//testReal:=BYTE_TO_REAL(arr_RcvData_Temp);
//数据接收处理
reciveFtrig(CLK:=receive1.busy);
IF reciveFtrig.Q THEN
	arr_RcvDataString:=arr_RcvDataStringTemp;
	arr_RcvDataStringTemp:=arr_RcvDataStringClear;
	RcvDataFlag:=TRUE;
	serialConnected:=TRUE;
END_IF
recTon(IN:=RcvDataFlag, PT:=T#20MS);
IF recTon.Q THEN
	RcvDataFlag:=FALSE;
END_IF
againSendS3(IN:=NOT RcvDataFlag,PT:=T#5S);
IF againSendS3.Q THEN
	sendstr:='S3$R';
	serialExcute:=TRUE;
	serialConnected:=FALSE;
	againSendS3(IN:=FALSE);
END_IF
IF TRUE THEN
	IF BYTE_TO_INT(arr_RcvDataString[4]-48)>0 THEN
		rec_ManulOrAuto:=TRUE;
		rec_MAStr:='Manul';
	ELSE
		rec_ManulOrAuto:=FALSE;
		rec_MAStr:='Auto';
	END_IF
	// 公式：(AD_CH6-LD_MIN)*(100/(LD_MAX-LD_MIN))
	AD_CH6:=CalMeth(arr_RcvDataString[28])*16*16+CalMeth(arr_RcvDataString[29])*16+CalMeth(arr_RcvDataString[30]);
	load:=(INT_TO_REAL(AD_CH6)-INT_TO_REAL(R00_LDMIN))*(100.0/(INT_TO_REAL(R01_LDMAX)-INT_TO_REAL(R00_LDMIN)));
	IF load>100.0 THEN
		load:=100.0;
		loadRunErr:=TRUE;
	END_IF
	IF load<0.0 THEN
		load:=0.0;
		loadRunErr:=TRUE;
	END_IF
	IF load<100.0 AND load>=0.0 THEN
		loadRunErr:=FALSE;
	END_IF
	// 公式：(AD_CH7-PH_MIN)*(100/(PH_MAX-PH_MIN))
	AD_CH7:=CalMeth(arr_RcvDataString[31])*16*16+CalMeth(arr_RcvDataString[32])*16+CalMeth(arr_RcvDataString[33]);	
	phase:=(INT_TO_REAL(AD_CH7)-INT_TO_REAL(R02_PHMIN))*(100.0/(INT_TO_REAL(R03_PHMAX)-INT_TO_REAL(R02_PHMIN)));
	IF phase>100.0 THEN
		phase:=100.0;
		phashRunErr:=TRUE;
	END_IF
	IF phase<0.0 THEN
		phase:=0.0;
		phashRunErr:=TRUE;
	END_IF
	IF phase<100.0 AND phase>=0.0 THEN
		phashRunErr:=FALSE;
	END_IF
END_IF
ACT_Send();
ACT_SetPreset();

ACTION ACT_Send:

CASE serialStep OF
	0:
	IF serialExcute THEN
		serialExcute:=FALSE;
		IF NOT serialBusy THEN
			serialStep:=90;
			serialBusy:=TRUE;
			serialDone:=FALSE;
			serialError:=FALSE;
			serialTimeOut:=FALSE;
			serialRecError:=FALSE;
		END_IF
	END_IF
	Timer1(IN:= FALSE);
	;
	10:
		arr_SendData:='SPL$R';
		send1(
			pSendData:= ADR(arr_SendData), 
			Length:=INT_TO_UDINT(LEN(arr_SendData)), 
			Busy=> , 
			Error=> , 
			TXbuffer:= gTxBuffer_SRF);
		serialStep:=serialStep+1;
	11:
		Timer1(IN:= NOT timer1.q, PT:=T#10MS);
		IF Timer1.Q THEN
			serialStep:=serialStep+1;
			Timer1(IN:= FALSE);
		END_IF
	12:
		Timer1(IN:= NOT timer1.q, PT:=T#500MS);
		IF Timer1.Q THEN
			serialStep:=6000;
			Timer1(IN:= FALSE);
			serialTimeOut:=TRUE;
			RETURN;
		END_IF
		IF NOT send1.busy AND NOT RcvDataFlag THEN
			Timer1(IN:= FALSE);
			serialTimeOut:=FALSE;
			serialStep:=serialStep+1;
		END_IF
		IF send1.Error <> COMERROR_NOERROR THEN
			serialRecError:=TRUE;
		END_IF
	13:
		Timer1(IN:= NOT timer1.q, PT:=T#50MS);
		IF Timer1.Q THEN
			serialStep:=90;
			Timer1(IN:= FALSE);
		END_IF
	90:
		arr_SendData:=sendstr;
		serialStep:=100;
	100:
		send1(
			pSendData:= ADR(arr_SendData), 
			Length:= INT_TO_UDINT(LEN(arr_SendData)), 
			Busy=> , 
			Error=> , 
			TXbuffer:= gTxBuffer_SRF);
		serialStep:=serialStep+10;
	110:
		Timer1(IN:= NOT timer1.q, PT:=T#10MS);
		IF Timer1.Q THEN
			serialStep:=serialStep+10;
			Timer1(IN:= FALSE);
		END_IF
	120:
		Timer1(IN:= NOT timer1.q, PT:=T#500MS);
		IF Timer1.Q THEN
			serialStep:=6000;
			Timer1(IN:= FALSE);
			serialTimeOut:=TRUE;
			RETURN;
		END_IF
		IF NOT send1.busy  THEN
			Timer1(IN:= FALSE);
			serialTimeOut:=FALSE;
			serialStep:=200;
		END_IF
		IF send1.Error <> COMERROR_NOERROR THEN
			serialRecError:=TRUE;
		END_IF
	200://数据处理
		serialStep:=serialStep+10;
	210:
		Timer1(IN:= NOT timer1.q, PT:=T#10MS);
		IF Timer1.Q THEN
			serialStep:=serialStep+10;
			Timer1(IN:= FALSE);
		END_IF
	220:
		//数据转换
		Timer1(IN:= FALSE);
		serialStep:=1000;
	
	1000:
		Timer1(IN:= NOT timer1.q, PT:=T#50MS);
		IF Timer1.Q THEN
			serialStep:=5000;
			Timer1(IN:= FALSE);
			// sendstr:='';
			serialTimeOut:=FALSE;
		END_IF
	;
	5000://done
		serialBusy:=FALSE;
		serialDone:=TRUE;
		serialError:=FALSE;
		serialStep:=0;
	;
	6000://error
		serialBusy:=FALSE;
		serialDone:=FALSE;
		serialError:=TRUE;
		serialStep:=0;
	;
	
END_CASE
END_ACTION

ACTION ACT_SetPreset:
CASE setPresetStep OF
	0:
	IF setPresetExt THEN
		setPresetExt:=FALSE;
		IF NOT setPresetBusy THEN
			setPresetStep:=100;
			setPresetBusy:=TRUE;
			setPresetDone:=FALSE;
			setPresetError:=FALSE;
		END_IF
	END_IF
	TimerSetPreset(IN:= FALSE);
	;
	100:
		decimalvalue:=LREAL_TO_INT(goPosLoad*10);
		decimalvalueP:=LREAL_TO_INT(goPosPhase*10);
		hexString:='';
		hexStringP:='';
		sendstr:='';
		IF goPosLoad>100 OR goPosLoad<0 OR goPosPhase>100 OR goPosPhase<0 THEN
			;
		ELSE
			IF goPosLoad=0 THEN
				hexString:='000';
			ELSE
				index:=(decimalvalue/256);
				hexString:=CONCAT(hexString,hexChars[index]);
				index:=((decimalvalue-index*256)/16);
				hexString:=CONCAT(hexString,hexChars[index]);
				index:=(decimalvalue MOD 16);
				hexString:=CONCAT(hexString,hexChars[index]);
			END_IF
			IF goPosPhase=0 THEN
				hexStringP:='000';
			ELSE
				index:=(decimalvalueP/256);
				hexStringP:=CONCAT(hexStringP,hexChars[index]);
				index:=((decimalvalueP-index*256)/16);
				hexStringP:=CONCAT(hexStringP,hexChars[index]);
				index:=(decimalvalueP MOD 16);
				hexStringP:=CONCAT(hexStringP,hexChars[index]);
			END_IF
			sendstr:=CONCAT(sendstr,'$$APGR');
			sendstr:=CONCAT(sendstr,hexString);
			sendstr:=CONCAT(sendstr,hexStringP);
			sendstr:=CONCAT(sendstr,'$R');
			serialExcute:=TRUE;
		END_IF
		setPresetStep:=setPresetStep+10;
	110:
		TimerSetPreset(IN:= TRUE,PT:=T#0.1S);
		IF TimerSetPreset.Q THEN
			TimerSetPreset(IN:= FALSE);
			setPresetStep:=setPresetStep+10;
		END_IF
	120:
		IF serialDone AND NOT serialBusy AND 
		ABS(load-goPosLoad)<0.5 AND ABS(phase-goPosPhase)<0.5 THEN
			setPresetStep:=setPresetStep+10;
		END_IF
		IF serialError THEN
			setPresetStep:=6000;
			RETURN;
		END_IF
	130:
		sendstr:='';
		sendstr:='P0$R';
		serialExcute:=TRUE;
		setPresetStep:=setPresetStep+10;
	140:
		TimerSetPreset(IN:= TRUE,PT:=T#0.03S);
		IF TimerSetPreset.Q THEN
			TimerSetPreset(IN:= FALSE);
			setPresetStep:=setPresetStep+10;
		END_IF
	150:
		IF serialDone THEN
			setPresetStep:=5000;
		END_IF
	
	5000://done
		setPresetBusy:=FALSE;
		setPresetDone:=TRUE;
		setPresetError:=FALSE;
		DataSave.fbDataSaveModule_EX_1.setLrealValue(FuncModule_RS232_SRF.goPosLoad,1);
		DataSave.fbDataSaveModule_EX_1.setLrealValue(FuncModule_RS232_SRF.goPosPhase,2);
		DataSave.fbDataSaveModule_EX_1.saveB:=TRUE;
		ups_CX51X0.Act_Wrtie();
		setPresetStep:=0;
	;
	6000://error
		setPresetBusy:=FALSE;
		setPresetDone:=FALSE;
		setPresetError:=TRUE;
		setPresetStep:=0;
	;
	
END_CASE
END_ACTION

METHOD CalASII_Str : STRING
VAR_INPUT
	date1:UINT;
END_VAR
IF date1=10 THEN
	CalASII_Str:='A';
END_IF
IF date1=11 THEN
	CalASII_Str:='B';
END_IF
IF date1=12 THEN
	CalASII_Str:='C';
END_IF
IF date1=13 THEN
	CalASII_Str:='D';
END_IF
IF date1=14 THEN
	CalASII_Str:='E';
END_IF
IF date1=15 THEN
	CalASII_Str:='F';
END_IF
IF date1<10 THEN
	CalASII_Str:=UINT_TO_STRING(date1);
END_IF
IF date1>15 THEN
	CalASII_Str:=UINT_TO_STRING(date1);
END_IF
END_METHOD

METHOD CalMeth : INT
VAR_INPUT
	byteIn:BYTE;
END_VAR
VAR_OUTPUT
	outInt:INT;
END_VAR
IF byteIn>=48 AND byteIn<=57 THEN
	outInt:=byteIn-48;
ELSE
	outInt:=byteIn-65+10;
END_IF
CalMeth:=outInt;
END_METHOD

METHOD LoadAndPhaseGo : BOOL
VAR_INPUT
	
END_VAR
VAR_OUTPUT
	
END_VAR
setPresetExt:=TRUE;
END_METHOD

METHOD LoadDEC : BOOL
VAR_INPUT
END_VAR
sendstr:='J84$R';
serialExcute:=true;
END_METHOD

METHOD LoadINC : BOOL
VAR_INPUT
END_VAR
sendstr:='J85$R';
serialExcute:=true;
END_METHOD

METHOD ManulORAuto : BOOL
VAR_INPUT
END_VAR
IF NOT rec_ManulOrAuto THEN
	sendstr:='M$R';
	serialExcute:=TRUE;
ELSE
	sendstr:='L$R';
	serialExcute:=TRUE;
END_IF
END_METHOD

METHOD PhaseDEC : BOOL
VAR_INPUT
END_VAR
sendstr:='J48$R';
serialExcute:=true;
END_METHOD

METHOD PhaseINC : BOOL
VAR_INPUT
END_VAR
sendstr:='J58$R';
serialExcute:=true;
END_METHOD

END_PROGRAM

// ---- POUs/Data/DownTimeRecordPOU.TcPOU
PROGRAM DownTimeRecordPOU
VAR
	fbGetCurTaskIndex:GetCurTaskIndex;
	nTaskNo:INT;
	tonPush:TON;
	tPush:TIME:=T#59.9S;
	fDownTime:REAL;
	fOtherDownTime:REAL;
	fOpDownTime:REAL;
END_VAR
VAR
	stPowerOnTime:ST_DownTimeRecord;// 记录上电运行总时间，从开始自动到结束自动的时间
	nPowerOnDay:UDINT:=0;// 记录上电天数

	stAutoRunTime:ST_DownTimeRecord;// 记录自动运行总时间，从开始自动到结束自动的时间
	AutoRunTime_temp:LREAL;// 缓存时间
	
	stManualMachineDownTime:ST_DownTimeRecord;// 记录手动状态下设备DownTime，
	ManualMachineDownTime_temp:LREAL;// 缓存时间
	
	stMachineDownTime:ST_DownTimeRecord;// 记录设备DownTime，从报错上升沿到下降沿
	MachineDownTime_temp:LREAL;// 缓存时间
	
	stOtherDownTime:ST_DownTimeRecord;// 记录设备其他DownTime，从暂停上升沿到下降沿
	OtherDownTime_temp:LREAL;// 缓存时间
	
	stOpLoadDownTime:ST_DownTimeRecord;// 记录设备操作员上料DownTime，从动作超时上升沿到下降沿
	OpLoadDownTime_Fix:LREAL;// 操作员固定时间
	OpLoadDownTime_temp:LREAL;// 缓存时间
	
	stOpUnloadDownTime:ST_DownTimeRecord;// 记录设备操作员下料DownTime，从动作超时上升沿到下降沿
	OpUnloadDownTime_Fix:LREAL;// 操作员固定时间
	OpUnloadDownTime_temp:LREAL;// 缓存时间
	
END_VAR


// 记录PLC上电总时间
	fbGetCurTaskIndex(index=>nTaskNo);
	IF TwinCAT_SystemInfoVarList._TaskInfo[nTaskNo].FirstCycle THEN// 上电初始时间
		stPowerOnTime.startTime:=TIME();
		nPowerOnDay:=0;
		stManualMachineDownTime.startTime:=TIME();
		ManualMachineDownTime_temp:=0;
		
		initState(stAutoRunTime);
		initState(stManualMachineDownTime);
		initState(stMachineDownTime);
		initState(stOtherDownTime);
		initState(stOpLoadDownTime);
		initState(stOpUnloadDownTime);
	END_IF
	stPowerOnTime.endTime:=TIME();
	calcTime(stPowerOnTime);
	
	stPowerOnTime.bMonitor:=((stPowerOnTime.start2end_s>=3600));// 监控的状态
	stPowerOnTime.rTrig(CLK:=stPowerOnTime.bMonitor);
	IF stPowerOnTime.rTrig.Q THEN// 累加1天
		stPowerOnTime.startTime:=TIME();
		nPowerOnDay:=nPowerOnDay+1;
	END_IF

// 记录自动运行总时间
	stAutoRunTime.rTrig(CLK:=gAutoRunningFlag);
	IF stAutoRunTime.rTrig.Q THEN// 注意，在初进入自动时同步 startTime 和 endTime
		// 此次是否需要初始化？
		(*initState(stAutoRunTime);
		initState(stMachineDownTime);
		initState(stOtherDownTime);
		initState(stOpLoadDownTime);
		initState(stOpUnloadDownTime);*)
		
		stAutoRunTime.startTime:=TIME();
		//
	END_IF
	stAutoRunTime.fTrig(CLK:=gAutoRunningFlag);
	IF stAutoRunTime.fTrig.Q THEN// 注意，在初进入自动时同步 startTime 和 endTime
		stManualMachineDownTime.startTime:=TIME();
		ManualMachineDownTime_temp:=0;
		
		stAutoRunTime.endTime:=TIME();
		calcTime(stAutoRunTime);
		AutoRunTime_temp:=0;
		stAutoRunTime.record_s:=stAutoRunTime.start2end_s;
		
		(*calcTime(stMachineDownTime);
		calcTime(stOtherDownTime);
		calcTime(stOpLoadDownTime);
		calcTime(stOpUnloadDownTime);
		stMachineDownTime.record_s:=stMachineDownTime.start2end_s;
		stOtherDownTime.record_s:=stOtherDownTime.start2end_s;
		stOpLoadDownTime.record_s:=stOpLoadDownTime.start2end_s;
		stOpUnloadDownTime.record_s:=stOpUnloadDownTime.start2end_s;*)
		// 做时间记录
		
		// 此次是否需要初始化？
		(*initState(stAutoRunTime);
		initState(stMachineDownTime);
		initState(stOtherDownTime);
		initState(stOpLoadDownTime);
		initState(stOpUnloadDownTime);*)
	END_IF


// 记录自动运行下: MachineDownTime 时间; OtherDownTime 时间; OpLoadDownTime 时间;  OpUnLoadDownTime 时间; 
	IF gAutoRunningFlag THEN// 自动状态下
	 (*MachineDownTime*) // 报错 上升沿-下降沿
		stMachineDownTime.bMonitor:=(gRunningState=RunningStatus.eErrorState);// 监控的状态
		stMachineDownTime.rTrig(CLK:=stMachineDownTime.bMonitor);
		IF stMachineDownTime.rTrig.Q THEN// 记录开始时间
			stMachineDownTime.startTime:=TIME();
			MachineDownTime_temp:=0;
		END_IF
		IF stMachineDownTime.bMonitor THEN
			stMachineDownTime.endTime:=TIME();
			calcTime(stMachineDownTime);
			MachineDownTime_temp:=(stMachineDownTime.start2end_s)-MachineDownTime_temp;// 获取每个扫描周期产生的时间差
			stMachineDownTime.record_s:=stMachineDownTime.record_s+MachineDownTime_temp;
			MachineDownTime_temp:=(stMachineDownTime.start2end_s);// 缓存最后一个扫描周期的总时长
		END_IF
		stMachineDownTime.fTrig(CLK:=stMachineDownTime.bMonitor);
		IF stMachineDownTime.fTrig.Q THEN// 记录结束状态
			stMachineDownTime.endTime:=TIME();
			calcTime(stMachineDownTime);
			MachineDownTime_temp:=0;
			// 做时间记录
				(*
				gDownTimeLog.append(CONCAT('DT,stMachineDownTime,',TO_STRING(stMachineDownTime.record_s)));
				*)
		END_IF
	 //
	 (*OtherDownTime*) // 暂停 上升沿-下降沿
		stOtherDownTime.bMonitor:=(gRunningState=RunningStatus.ePauseState);// 监控的状态
		stOtherDownTime.rTrig(CLK:=stOtherDownTime.bMonitor);
		IF stOtherDownTime.rTrig.Q THEN// 记录开始时间
			stOtherDownTime.startTime:=TIME();
			OtherDownTime_temp:=0;
		END_IF
		IF stOtherDownTime.bMonitor THEN
			stOtherDownTime.endTime:=TIME();
			calcTime(stOtherDownTime);
			OtherDownTime_temp:=(stOtherDownTime.start2end_s)-OtherDownTime_temp;// 获取每个扫描周期产生的时间差
			stOtherDownTime.record_s:=stOtherDownTime.record_s+OtherDownTime_temp;
			OtherDownTime_temp:=(stOtherDownTime.start2end_s);// 缓存最后一个扫描周期的总时长
		END_IF
		stOtherDownTime.fTrig(CLK:=stOtherDownTime.bMonitor);
		IF stOtherDownTime.fTrig.Q THEN// 记录结束状态
			stOtherDownTime.endTime:=TIME();
			calcTime(stOtherDownTime);
			OtherDownTime_temp:=0;
			// 做时间记录
				(*
				gDownTimeLog.append(CONCAT('DT,stOtherDownTime,',TO_STRING(stOtherDownTime.record_s)));
				*)
		END_IF
	 //
	 (*OpLoadDownTime*) //  上升沿-下降沿
	 	// 此处不会记录第一次进入自动时，OP不上料的情况
//		stOpLoadDownTime.rTrig(CLK:=L_Robot_Load.Can_Getting_DUT);//(CLK:=L_Robot_Load.Getting_DUT);
//		IF stOpLoadDownTime.rTrig.Q OR (gRunningState<>RunningStatus.eAutoState) THEN// 记录开始时间
//			stOpLoadDownTime.startTime:=TIME();
//			OpLoadDownTime_temp:=0;
//			stOpLoadDownTime.bMonitor:=TRUE;
//		END_IF
//		IF stOpLoadDownTime.bMonitor THEN
//			stOpLoadDownTime.endTime:=TIME();
//			calcTime(stOpLoadDownTime);
//			OpLoadDownTime_Fix:=3;// 常数, 按实际情况配置------------------------------------------------------------------------------
//			IF (stOpLoadDownTime.start2end_s>OpLoadDownTime_Fix) THEN
//				OpLoadDownTime_temp:=(stOpLoadDownTime.start2end_s(*-OpLoadDownTime_Fix*))-OpLoadDownTime_temp;// 获取每个扫描周期产生的时间差
//				stOpLoadDownTime.record_s:=stOpLoadDownTime.record_s+OpLoadDownTime_temp;
//				OpLoadDownTime_temp:=(stOpLoadDownTime.start2end_s(*-OpLoadDownTime_Fix*));// 缓存最后一个扫描周期的总时长
//			END_IF
//		END_IF
//		stOpLoadDownTime.fTrig(CLK:=L_Robot_Load.Can_Getting_DUT);
//		IF stOpLoadDownTime.fTrig.Q THEN// 记录结束状态
//			stOpLoadDownTime.bMonitor:=FALSE;
//			stOpLoadDownTime.endTime:=TIME();
//			calcTime(stOpLoadDownTime);
//			OpLoadDownTime_temp:=0;// 清除缓存时间
//			// 做时间记录
//				(*
//				gDownTimeLog.append(CONCAT('DT,stOpLoadDownTime,',TO_STRING(stOpLoadDownTime.record_s)));
//				*)
//		END_IF
//	 //
//	 (*OpUnLoadDownTime*) //  上升沿-下降沿
//		stOpUnloadDownTime.bMonitor:=gStationUnLoad.I_BeltEndisHaveDutSensor_1 OR gStationUnLoad.I_BeltEndisHaveDutSensor_2;// 监控的状态
//		stOpUnloadDownTime.rTrig(CLK:=stOpUnloadDownTime.bMonitor);
//		IF stOpUnloadDownTime.rTrig.Q OR (gRunningState<>RunningStatus.eAutoState) THEN// 记录开始时间
//			stOpUnloadDownTime.startTime:=TIME();
//			OpUnloadDownTime_temp:=0;
//		END_IF
//		IF stOpUnloadDownTime.bMonitor THEN
//			stOpUnloadDownTime.endTime:=TIME();
//			calcTime(stOpUnloadDownTime);
//			OpUnloadDownTime_Fix:=3;// 常数, 按实际情况配置------------------------------------------------------------------------------
//			IF (stOpUnloadDownTime.start2end_s>OpUnloadDownTime_Fix) THEN
//				OpUnloadDownTime_temp:=(stOpUnloadDownTime.start2end_s(*-OpUnloadDownTime_Fix*))-OpUnloadDownTime_temp;// 获取每个扫描周期产生的时间差
//				stOpUnloadDownTime.record_s:=stOpUnloadDownTime.record_s+OpUnloadDownTime_temp;
//				OpUnloadDownTime_temp:=(stOpUnloadDownTime.start2end_s(*-OpUnloadDownTime_Fix*));// 缓存最后一个扫描周期的总时长
//			END_IF
//		END_IF
//		stOpUnloadDownTime.fTrig(CLK:=stOpUnloadDownTime.bMonitor);
//		IF stOpUnloadDownTime.fTrig.Q THEN// 记录结束状态
//			stOpUnloadDownTime.endTime:=TIME();
//			calcTime(stOpUnloadDownTime);
//			OpUnloadDownTime_temp:=0;// 清除缓存时间
//			// 做时间记录
//				(*
//				gDownTimeLog.append(CONCAT('DT,stOpUnloadDownTime,',TO_STRING(stOpUnloadDownTime.record_s)));
//				*)
//		END_IF
//	 //
	ELSE// 手动状态下
		stManualMachineDownTime.endTime:=TIME();
		calcTime(stManualMachineDownTime);
		ManualMachineDownTime_temp:=(stManualMachineDownTime.start2end_s)-ManualMachineDownTime_temp;// 获取每个扫描周期产生的时间差
		stManualMachineDownTime.record_s:=stManualMachineDownTime.record_s+ManualMachineDownTime_temp;
		ManualMachineDownTime_temp:=(stManualMachineDownTime.start2end_s);// 缓存最后一个扫描周期的总时长
	END_IF

// 定时上报
tonPush(IN:=NOT tonPush.Q,PT:=tPush);
IF tonPush.Q THEN
	IF gAutoRunningFlag THEN
		stAutoRunTime.endTime:=TIME();
		calcTime(stAutoRunTime);
		AutoRunTime_temp:=0;
		stAutoRunTime.record_s:=stAutoRunTime.start2end_s;
//		gPowerONTotalTime:=gPowerONTotalTime+1;
	END_IF
	fDownTime:=TO_REAL(stManualMachineDownTime.record_s+stMachineDownTime.record_s);
	fOtherDownTime:=TO_REAL(stOtherDownTime.record_s);
	fOpDownTime:=TO_REAL(stOpLoadDownTime.record_s+stOpUnloadDownTime.record_s);
	
	//(*
	gDownTimeLog.append(CONCAT('DT,stAutoRunTime,',TO_STRING(stAutoRunTime.record_s)));
	gDownTimeLog.append(CONCAT('DT,stManualMachineDownTime,',TO_STRING(stManualMachineDownTime.record_s)));
	gDownTimeLog.append(CONCAT('DT,stMachineDownTime,',TO_STRING(stMachineDownTime.record_s)));
	gDownTimeLog.append(CONCAT('DT,stOtherDownTime,',TO_STRING(stOtherDownTime.record_s)));
//	gDownTimeLog.append(CONCAT('DT,stOpLoadDownTime,',TO_STRING(stOpLoadDownTime.record_s)));
//	gDownTimeLog.append(CONCAT('DT,stOpUnloadDownTime,',TO_STRING(stOpUnloadDownTime.record_s)));
	//*)
	// 此次需要做发送给上位机的逻辑
//	PLC_SW1.appendSend(0,0,80,0.0,TO_REAL(stManualMachineDownTime.record_s),0.0,TO_REAL(stOtherDownTime.record_s),0.0,gErrIDToSW,'');
	
	// 记录完毕清除数据，重新记录
	initState(stAutoRunTime);
	initState(stManualMachineDownTime);
	initState(stMachineDownTime);
	initState(stOtherDownTime);
	initState(stOpLoadDownTime);
	initState(stOpUnloadDownTime);
	AutoRunTime_temp:=0;
	ManualMachineDownTime_temp:=0;
	MachineDownTime_temp:=0;
	OpLoadDownTime_temp:=0;
	OpUnloadDownTime_temp:=0;
END_IF

METHOD calcTime : BOOL
VAR_IN_OUT
	stDownTimeRecord:ST_DownTimeRecord;
END_VAR

stDownTimeRecord.start2end_time:=(stDownTimeRecord.endTime-stDownTimeRecord.startTime);
stDownTimeRecord.start2end_ms:=TO_UDINT(stDownTimeRecord.endTime-stDownTimeRecord.startTime);
stDownTimeRecord.start2end_s:=TO_LREAL(stDownTimeRecord.start2end_ms)*0.001;
//stDownTimeRecord.startTime:=stDownTimeRecord.endTime;

calcTime:=TRUE;
END_METHOD

METHOD initState : BOOL
VAR_IN_OUT
	stDownTimeRecord:ST_DownTimeRecord;
END_VAR

stDownTimeRecord.bMonitor:=FALSE;
stDownTimeRecord.startTime:=stDownTimeRecord.endTime:=TIME();
stDownTimeRecord.start2end_ms:=0;
stDownTimeRecord.start2end_s:=0;
stDownTimeRecord.start2end_time:=TO_TIME(0);
stDownTimeRecord.record_s:=0;
stDownTimeRecord.rTrig(CLK:=FALSE);
stDownTimeRecord.fTrig(CLK:=FALSE);

initState:=TRUE;
END_METHOD

END_PROGRAM

// ---- POUs/Data/FB_WStringSave.TcPOU
PROGRAM FB_WStringSave
VAR CONSTANT
	Maxlenght:INT:=100;
END_VAR

VAR_INPUT
	filter:WSTRING:=",";
	readTrig:BOOL;
	writeTrig:BOOL;
	savePath : T_MaxString;
END_VAR
VAR_OUTPUT
	nErrorId : UDINT;
	bError : BOOL;
	readDone:BOOL;
	saveDone:BOOL;
	readError:BOOL;
	saveError:BOOL;
END_VAR
VAR
	fbFileOpen:FB_FILEOPEN;
	fbFileClose:FB_FILECLOSE;
	fbFileGet:FB_FILEGETS;
	fbFilePut:FB_FILEPUTS;
	fbWriter:FB_FILEWRITE;

	hFile : UINT;
	sReadLine : T_MaxString;
	wsWriteLine : WSTRING(255); 
	sWriteLine : T_MaxString;
	wsReadLine : WSTRING(255);
	wsReadTemp : WSTRING(255);
	itemp:INT;
	inputArry: ARRAY [1..Maxlenght] OF WSTRING;
	outputArry: ARRAY [1..Maxlenght] OF WSTRING;
	findposstart	:INT;
	findposend		:INT;
	find_pos		:INT;
	recStrTemp		:WSTRING(255);
	nReadStep : UINT;
	nWriteStep : UINT;
END_VAR

readDone:=FALSE;
fbFileOpen(
	sNetId:= , 
	sPathName:= , 
	nMode:= , 
	ePath:= , 
	bExecute:= , 
	tTimeout:= , 
	bBusy=> , 
	bError=> , 
	nErrId=> , 
	hFile=>hFile );
	
fbFileClose(
	sNetId:= , 
	hFile:= hFile, 
	bExecute:= , 
	tTimeout:= , 
	bBusy=> , 
	bError=> , 
	nErrId=> );

fbFileGet(
	sNetId:= , 
	hFile:= hFile, 
	bExecute:= , 
	tTimeout:= , 
	bBusy=> , 
	bError=> , 
	nErrId=> , 
	sLine=> , 
	bEOF=> );
	
fbFilePut(
	sNetId:= , 
	hFile:= hFile, 
	sLine:= , 
	bExecute:= , 
	tTimeout:= , 
	bBusy=> , 
	bError=> , 
	nErrId=> );
IF readTrig THEN
	nReadStep:=10;
	readTrig:=FALSE;
END_IF
IF writeTrig THEN
	nWriteStep:=10;
	writeTrig:=FALSE;
END_IF
Act_Read();
Act_Write();

ACTION Act_Read:
CASE nReadStep OF
	0:
	;
	10:
		//复位状态
		bError := FALSE;
		nErrorId := 0;
		fbFileopen(bExecute:= FALSE);
		fbFileclose(bExecute:= FALSE);
		fbFileGet(bExecute:= FALSE);
		readError:=FALSE;
		nReadStep := 20;
		fbFileopen(sNetId:= , sPathName:= savePath,ePath:= PATH_GENERIC, bExecute:= TRUE, nMode:=FOPEN_MODEREAD ,hFile=>hFile );
	20:	
		IF NOT fbFileopen.bBusy THEN
			fbFileopen(bExecute:= FALSE);
			IF fbFileopen.bError THEN//出错
				bError := TRUE;
				nErrorId := fbFileopen.nErrId;
				nReadStep := 200;
				readError:=TRUE;
			ELSE //正常
				
				nReadStep := 30;
			
			END_IF
		END_IF
	30:
		nReadStep := 40;
	40:
		nReadStep := 100;
	100:
		fbFileGet(hFile:= hFile, bExecute:= TRUE, sLine=>sReadLine);
		UTF8_TO_WSTRING(ADR(wsReadLine),ADR(sReadLine),SIZEOF(sReadLine));
		IF NOT fbFileGet.bBusy THEN
			fbFileGet(bExecute:= FALSE);
			IF fbFileGet.bError THEN//出错
				bError := TRUE;
				nErrorId := fbFileGet.nErrId;
				nReadStep := 200;
				readError:=TRUE;
			ELSE //正常
				IF NOT fbFileGet.bEOF THEN //继续读取
					nReadStep := 110;
				ELSE
					//读取完成
					nReadStep := 110;
				END_IF
				
				
			
			END_IF
		END_IF
		
	110:
		wsReadTemp:=wsReadLine;
		ReadToOut();
		nReadStep := 200;		
		;
	200:
		fbFileClose( hFile:= hFile, bExecute:= TRUE ,nErrId=> );
		IF NOT fbFileClose.bBusy THEN
			fbFileClose(bExecute:= FALSE);
			IF fbFileClose.bError THEN//出错
				bError := TRUE;
				nErrorId := fbFileClose.nErrId;
				nReadStep := 1000;
			ELSE //正常
				
				nReadStep := 2000;
			
			END_IF
		END_IF
		
	1000:
		//报错
		nReadStep := 0;
		
	2000:
		//完成
		nReadStep := 0;
		readDone:=TRUE;
END_CASE
END_ACTION

ACTION Act_Write:
CASE nWriteStep OF
	0:
	;
	10:
		//复位状态
		bError := FALSE;
		nErrorId := 0;
		fbFileOpen(bExecute:= FALSE);
		fbFileClose(bExecute:= FALSE);
		fbFilePut(bExecute:= FALSE);
		saveError:=FALSE;
		nWriteStep := 20;
	20:
		fbFileOpen(sNetId:= , sPathName:= savePath, nMode:= FOPEN_MODEWRITE, ePath:= , bExecute:= TRUE,hFile=>hFile );		
		IF NOT fbFileOpen.bBusy THEN
			fbFileOpen(bExecute:= FALSE);
			IF fbFileOpen.bError THEN//出错
				bError := TRUE;
				nErrorId := fbFileOpen.nErrId;
				nWriteStep := 200;
				saveError:=TRUE;
			ELSE //正常
				
				nWriteStep := 100;
			
			END_IF
		END_IF

	100:
		InToWrite();
		nWriteStep := 110;
	110:
		WSTRING_TO_UTF8(ADR(sWriteLine),ADR(wsWriteLine),SIZEOF(wsWriteLine));
		fbFilePut(hFile:= hFile, bExecute:= TRUE, sLine:=sWriteLine);
		
		IF NOT fbFilePut.bBusy THEN
			fbFilePut(bExecute:= FALSE);
			IF fbFilePut.bError THEN//出错
				bError := TRUE;
				nErrorId := fbFilePut.nErrId;
				nWriteStep := 200;
				saveError:=TRUE;
			ELSE //正常
				//写入完成
				nWriteStep := 200;	
			END_IF
		END_IF
		wsWriteLine:="";
				
		;
	200:
		fbFileClose( hFile:= hFile, bExecute:= TRUE ,nErrId=> );
		IF NOT fbFileClose.bBusy THEN
			fbFileClose(bExecute:= FALSE);
			IF fbFileClose.bError THEN//出错
				bError := TRUE;
				nErrorId := fbFileClose.nErrId;
				nWriteStep := 1000;
				saveError:=TRUE;
			ELSE //正常
				
				nWriteStep := 2000;
			
			END_IF
		END_IF
		
	1000:
		//报错
		nWriteStep := 0;
		
	2000:
		//完成
		nWriteStep := 0;
		
END_CASE
END_ACTION

METHOD getWString : BOOL
VAR_IN_OUT
	value:WSTRING;
END_VAR
VAR_INPUT
	num:UDINT;
END_VAR
IF 0<=num AND UDINT_TO_INT(num)<=Maxlenght THEN
	value:=outputArry[num];
	getWString:=TRUE;
ELSE
	value:="";
	getWString:=FALSE;
END_IF
END_METHOD

ACTION InToWrite:
FOR itemp:=1 TO Maxlenght DO
	wsWriteLine:=WCONCAT(wsWriteLine,inputArry[itemp]);
	wsWriteLine:=WCONCAT(wsWriteLine,filter);
END_FOR
END_ACTION

ACTION ReadToOut:
FOR itemp:=1 TO Maxlenght DO
	find_pos:=wFIND(wsReadTemp, filter);
	IF find_pos>0 THEN
		findposstart:=find_pos;
		outputArry[itemp]:=WMID(wsReadTemp,find_pos-1,1);
		wsReadTemp:=WDELETE(wsReadTemp,find_pos,1);
		find_pos:=0;
	END_IF
END_FOR
END_ACTION

METHOD setWString : BOOL
VAR_INPUT
	value:WSTRING;
END_VAR
VAR_INPUT
	num:UDINT;
END_VAR
IF 0<=num AND uDINT_TO_INT(num)<=Maxlenght THEN
	inputArry[num]:=value;
	setWString:=TRUE;
ELSE
	setWString:=FALSE;
END_IF
END_METHOD

END_PROGRAM

// ---- POUs/IO/TesterIO.TcPOU
{attribute'TcContextName':='IOTask'}
PROGRAM TesterIO
VAR
	fbIOBase_Input:FB_IOBase_Input_New;//工站1 Input 
	
	fbIOBase_Output:FB_IOBase_Output_New;//工站1 Output 
	 
	DOE_DOE1IO AT%I*:UDINT;
	DOE_DOE2IO AT%I*:UDINT;

	I_Handle1FixVacuum2Ext: INT;
	I_Handle1FixVacuum1Ext: INT;
END_VAR


//工站1 Input 
	fbIOBase_Input(
		iIOModuleNum:= 5, 
		iLanguage:= TO_UINT(gCNErrShow), //TO_UINT(gCNErrShow)
		sFileName:= 'C:\IOFilePath\Input1.csv', 
		bReload:= , 
		stIOBase=> );


//工站1 Output 
	fbIOBase_Output(
		iIOModuleNum:= 5, 
		stIOBase:= , 
		iLanguage:= TO_UINT(gCNErrShow), //TO_UINT(gCNErrShow)
		sFileName:= 'C:\IOFilePath\Output1.csv', 
		bReload:= );




//输入映射---映射到程序内部变量
ACT_Input();//工站1 Input 


//输出映射---映射到程序内部变量
ACT_Output();//工站1 Output 


// 通讯IO
ACT_Communication();

ACTION ACT_Communication:
FuncModule_RS232_TBP(
	noRotation=> gICP.TruboPumNoRotation, 
	brake=> gICP.TruboPumDcc, 
	acc=> gICP.TruboPumAcc, 
	atTagetSpeed=> gICP.TruboPumNormal, 
	alarm=> gICP.TruboPumAlarm, 
	remote=> gICP.TruboPumRemote, 
	failure=> gICP.TruboPumError, 
	rotationSpeed=> gICP.TruboPumRotationSpeed, 
	tMSTemperature=> gICP.TruboPumTMS);
END_ACTION

ACTION ACT_Input:
//(*驱动器DI 映射*)
//********************上料电机

//gLoad_AXIS.I_X1NLimit:=Load_X1IO.19;
//gLoad_AXIS.I_X1Home:=Load_X1IO.20;
//gLoad_AXIS.I_X1PLimit:=Load_X1IO.18;


//********************载具电机

//gTestSocket_AXIS.I_X1NLimit:=TestSocket_X1IO.18;
//gTestSocket_AXIS.I_X1Home:=TestSocket_X1IO.16;
//gTestSocket_AXIS.I_X1PLimit:=TestSocket_X1IO.17;

//gRXTest_AXIS.I_CY3NLimit:=RXTest_CY3IO.19;
//gRXTest_AXIS.I_CY3Home:=RXTest_CY3IO.22;
//gRXTest_AXIS.I_CY3PLimit:=RXTest_CY3IO.18;

//********************TX电机***********
////*******此处为量产660系列映射地址
//gTXTest_Axis.I_Y1NLimit:=TXTest_Y1IO.17;
//gTXTest_Axis.I_Y1Home:=TXTest_Y1IO.18;
//gTXTest_Axis.I_Y1PLimit:=TXTest_Y1IO.16;

/////////以下为临时应用 采用620驱动器///
//gTXTest_Axis.I_Y1NLimit:=TXTest_Y1IO.21;
//gTXTest_Axis.I_Y1Home:=TXTest_Y1IO.18;
//gTXTest_Axis.I_Y1PLimit:=TXTest_Y1IO.20;

//********************机台IO
//////模块1
//gDOE_AXIS.I_DOE2PLimit:=fbIOBase_Input.stIOBase[1].io[1]; //启动
//gDOE_AXIS.I_DOE2NLimit:=fbIOBase_Input.stIOBase[1].io[2]; //停止
//gMachineUtility.I_Reset:=fbIOBase_Input.stIOBase[1].io[3]; //复位
//gMachineUtility.I_EStop:=fbIOBase_Input.stIOBase[1].io[4] ; //急停
////:=fbIOBase_Input.stIOBase[1].io[5] ; //备用

////:=fbIOBase_Input.stIOBase[1].io[8] ; //备用
//gMachineUtility.I_PressureDetection1:=fbIOBase_Input.stIOBase[1].io[9] ; //气压检测

//gMachineUtility.I_SafeDoor_1:=fbIOBase_Input.stIOBase[1].io[13]; //安全门
//gMachineUtility.I_SafeDoor_2:=fbIOBase_Input.stIOBase[1].io[14]; //安全门
//gMachineUtility.I_SafeDoor_3:=fbIOBase_Input.stIOBase[1].io[15]; //安全门
//gMachineUtility.I_SafeDoor_4:=fbIOBase_Input.stIOBase[1].io[16]; //安全门


gICP.LiftPinExtSensor:=fbIOBase_Input.stIOBase[1].io[1]; //Lift UP
gICP.LiftPinRetSensor:=fbIOBase_Input.stIOBase[1].io[2]; //Lift Down
gICP.ElectrodeCylExtSensor:=fbIOBase_Input.stIOBase[1].io[3] AND fbIOBase_Input.stIOBase[1].io[4] AND fbIOBase_Input.stIOBase[1].io[14] AND fbIOBase_Input.stIOBase[1].io[15]; //Eletrode UP1 AND UP2
gICP.ElectrodeCylRetSensor:=fbIOBase_Input.stIOBase[1].io[5] AND fbIOBase_Input.stIOBase[1].io[6] AND fbIOBase_Input.stIOBase[1].io[16] AND fbIOBase_Input.stIOBase[2].io[1] ; //Eletrode Down1 AND Down2
gICP.GateDoorExtSensor:=fbIOBase_Input.stIOBase[1].io[7]; //GateDoor open
gICP.GateDoorRetSensor:=fbIOBase_Input.stIOBase[1].io[8]; //GateDoor Close
gICP.I_ARMHome:=fbIOBase_Input.stIOBase[1].io[9]; //ARM IN Sensor
gICP.I_LLSwitch:=fbIOBase_Input.stIOBase[1].io[10]; // LoadLock Switch Sensor
gICP.I_WaferCheck:=fbIOBase_Input.stIOBase[1].io[11]; //WaferCheck Sensor
gICP.PDVOpenSensor:=fbIOBase_Input.stIOBase[1].io[12]; //PDVOpen Sensor
gICP.PDVCloseSensor:=fbIOBase_Input.stIOBase[1].io[13]; //PDVClose Sensor
//gICP.PDV:=fbIOBase_Input.stIOBase[1].io[13]; //WaferCheck Sensor
//gICP.TruboPumAcc:=fbIOBase_Input.stIOBase[1].io[15]; // TruboPumAcc
//gICP.TruboPumDcc:=fbIOBase_Input.stIOBase[1].io[16]; // TruboPumDcc
//gICP.TruboPumNormal:=fbIOBase_Input.stIOBase[2].io[1]; // TruboPumNormal
gICP.I_ATMSensor:=fbIOBase_Input.stIOBase[2].io[2]; // ATMSensor
gICP.MachianicalPumAcc:=fbIOBase_Input.stIOBase[2].io[3]; // I_MP Start
gICP.MachianicalPumAlm:=fbIOBase_Input.stIOBase[2].io[4]; // I_MP Failure

gICP.PowerRF_Alrm:=fbIOBase_Input.stIOBase[2].io[5]; // 600W
gICP.SourceRF_Alrm:=fbIOBase_Input.stIOBase[2].io[6]; // 2000W
gICP.PowerRF_ON:=fbIOBase_Input.stIOBase[2].io[7]; // 600W
gICP.SourceRF_ON:=fbIOBase_Input.stIOBase[2].io[8]; // 2000W

 
gICP.I_WaterTemperatureCheck:=fbIOBase_Input.stIOBase[2].io[9]; 
gICP.I_WaterFlowCheck:=fbIOBase_Input.stIOBase[2].io[10];
gICP.I_PressureCheck:=fbIOBase_Input.stIOBase[2].io[11]; 
gICP.HeCheckGaugeReal:=PLC_HeliumPressure.bRecReal;
END_ACTION

ACTION ACT_Output:

//(*IO模块 映射*)
//模块1
fbIOBase_Output.stIOBase[1].io[1]:=gICP.ForlinLineValveExtRelay;
fbIOBase_Output.stIOBase[1].io[2]:=gICP.ISOExtRelay;
fbIOBase_Output.stIOBase[1].io[3]:=gICP.RoughValveExtRelay;
fbIOBase_Output.stIOBase[1].io[4]:=gICP.VentExtRelay;
fbIOBase_Output.stIOBase[1].io[5]:=gICP.SlowPummingExtRelay;
fbIOBase_Output.stIOBase[1].io[6]:=gICP.FastPummingExtRelay;
fbIOBase_Output.stIOBase[1].io[7]:=gICP.LiftPinRetRelay;
fbIOBase_Output.stIOBase[1].io[8]:=gICP.LiftPinExtRelay;
fbIOBase_Output.stIOBase[1].io[9]:=gICP.ElectrodeCylRetRelay;
fbIOBase_Output.stIOBase[1].io[10]:=gICP.ElectrodeCylExtRelay;
fbIOBase_Output.stIOBase[1].io[11]:=gICP.AIMExtRelay;
fbIOBase_Output.stIOBase[1].io[12]:=gICP.HeINExtRelay;
fbIOBase_Output.stIOBase[1].io[13]:=gICP.HePumExtRelay;
fbIOBase_Output.stIOBase[1].io[14]:=gICP.PDVOpenRelay;
fbIOBase_Output.stIOBase[1].io[15]:=gICP.PDVCloseRelay;
//fbIOBase_Output.stIOBase[1].io[16]:=gICP.PowerRFOpenRelay;
//模块2
fbIOBase_Output.stIOBase[2].io[1]:=gICP.MachianicalPumOpen;
//fbIOBase_Output.stIOBase[2].io[2]:=gICP.MachianicalPumOpen;// reset

fbIOBase_Output.stIOBase[2].io[3]:=gICP.GateDoorExtRelay;
fbIOBase_Output.stIOBase[2].io[4]:=gICP.GateDoorRetRelay;
//fbIOBase_Output.stIOBase[2].io[5]:=gICP.TruboPumOpen;
//fbIOBase_Output.stIOBase[2].io[6]:=gICP.TruboPumOpen;
//fbIOBase_Output.stIOBase[2].io[5]:=gICP.PowerRFResetRelay;
//fbIOBase_Output.stIOBase[2].io[6]:=gICP.SourceRFResetRelay;
//fbIOBase_Output.stIOBase[2].io[7]:=gICP.TruboPumReset;
fbIOBase_Output.stIOBase[2].io[8]:=gICP.SourceRFOpenRelay;
fbIOBase_Output.stIOBase[2].io[9]:=gICP.GVA1ExtRelay;
fbIOBase_Output.stIOBase[2].io[10]:=gICP.GVA2ExtRelay;
fbIOBase_Output.stIOBase[2].io[11]:=gICP.GVA3ExtRelay;
fbIOBase_Output.stIOBase[2].io[12]:=gICP.GVA4ExtRelay;
fbIOBase_Output.stIOBase[2].io[13]:=gICP.GVA5ExtRelay;
fbIOBase_Output.stIOBase[2].io[14]:=gICP.GVA6ExtRelay;
fbIOBase_Output.stIOBase[2].io[15]:=gICP.GVA7ExtRelay;
fbIOBase_Output.stIOBase[2].io[16]:=gICP.GVA8ExtRelay;

fbIOBase_Output.stIOBase[3].io[1]:=gICP.GVB1ExtRelay;
fbIOBase_Output.stIOBase[3].io[2]:=gICP.GVB2ExtRelay;
fbIOBase_Output.stIOBase[3].io[3]:=gICP.GVB3ExtRelay;
fbIOBase_Output.stIOBase[3].io[4]:=gICP.GVB4ExtRelay;
fbIOBase_Output.stIOBase[3].io[5]:=gICP.GVB5ExtRelay;
fbIOBase_Output.stIOBase[3].io[6]:=gICP.GVB6ExtRelay;
fbIOBase_Output.stIOBase[3].io[7]:=gICP.GVB7ExtRelay;
fbIOBase_Output.stIOBase[3].io[8]:=gICP.GVB8ExtRelay;
fbIOBase_Output.stIOBase[3].io[9]:=gICP.GVA9ExtRelay;
fbIOBase_Output.stIOBase[3].io[10]:=gICP.GVB9ExtRelay;
fbIOBase_Output.stIOBase[3].io[11]:=gICP.GVA10ExtRelay_Vent;
fbIOBase_Output.stIOBase[3].io[12]:=gICP.GV20ExtRelay_Main;
END_ACTION

END_PROGRAM

// ---- POUs/BaseModule/IO/FB_IOBase_Input_New.TcPOU
FUNCTION_BLOCK FB_IOBase_Input_New
VAR CONSTANT
	MAX_IO_MODULE_NUM:DINT:=15;
END_VAR
VAR_INPUT
	iIOModuleNum:DINT;//输入输出模块数量
	iLanguage:UINT;//0：英文；1：中文
	sFileName:T_MaxString:='C:\IOFilePath\iocsvfile.csv';//'Hard Disk\IOFilePath\iocsvfile.csv'
	bReload:BOOL;//加载配置文件 触发
END_VAR
VAR_OUTPUT
	stIOBase:ARRAY [1..MAX_IO_MODULE_NUM] OF ST_INPUT_IO;
END_VAR
VAR
	HMIITF:ST_IOBase_Show_HMI;
	
	iIOModuleNum_Temp:DINT;//输入输出模块数量
	
	next_R_TRIG:R_TRIG;
	back_R_TRIG:R_TRIG;
	targer_R_TRIG:R_TRIG;
	
	iCurrPage:DINT:=1;
	iIndex_1:DINT;
	iIndex_2:DINT;
	
	readBuff:ARRAY [1..MAX_IO_MODULE_NUM*16] OF ST_DataFmtBase;
	fbFileReadWrite:FB_IOFileReadWrite;
	bInit:BOOL;
	bRefresh:BOOL;
	Refresh_R_TRIG:R_TRIG;
	iLanguage_temp:UINT;//0：英文；1：中文
END_VAR


HMIITF.sIOType:='Input';

iIOModuleNum_Temp:=iIOModuleNum;
IF iIOModuleNum<0 THEN
	iIOModuleNum_Temp:=0;
ELSIF iIOModuleNum>MAX_IO_MODULE_NUM THEN
	iIOModuleNum_Temp:=MAX_IO_MODULE_NUM;
END_IF

(*HMI process*)
 (* Next button *)
	next_R_TRIG(CLK:=HMIITF.bNextPage);
	IF next_R_TRIG.Q THEN
		iCurrPage:=iCurrPage+1;
		bRefresh:=TRUE;
	END_IF
 (* Back button *)
	back_R_TRIG(CLK:=HMIITF.bBackPage);
	IF back_R_TRIG.Q THEN
		iCurrPage:=iCurrPage-1;
		bRefresh:=TRUE;
	END_IF
 (* Targer button *)
 	IF HMIITF.iTargerPage<=0 THEN
		HMIITF.iTargerPage:=iIOModuleNum_Temp;
	ELSIF HMIITF.iTargerPage>iIOModuleNum_Temp THEN
		HMIITF.iTargerPage:=1;
	END_IF
	targer_R_TRIG(CLK:=HMIITF.bTargerPage);
	IF targer_R_TRIG.Q THEN
		iCurrPage:=HMIITF.iTargerPage;
		bRefresh:=TRUE;
	END_IF

	IF iCurrPage<=0 THEN
		iCurrPage:=iIOModuleNum_Temp;
	ELSIF iCurrPage>iIOModuleNum_Temp THEN
		iCurrPage:=1;
	END_IF
	HMIITF.iCurrPage:=iCurrPage;
	HMIITF.iMaxPage:=iIOModuleNum_Temp;
	
	FOR iIndex_1:=1 TO 16 BY 1 DO
		HMIITF.bIO[iIndex_1]:=stIOBase[iCurrPage].io[iIndex_1];//IO状态映射
	END_FOR
	IF bRefresh THEN
		FOR iIndex_1:=1 TO 16 BY 1 DO
			HMIITF.bIO[iIndex_1]:=stIOBase[iCurrPage].io[iIndex_1];//IO状态映射
			
			CASE iLanguage OF
				0:
					FOR iIndex_2:=1 TO (MAX_IO_MODULE_NUM*16) BY 1 DO
						IF iCurrPage=readBuff[iIndex_2].nGroup AND iIndex_1=readBuff[iIndex_2].nNumber THEN
							HMIITF.sInfor[iIndex_1]:=TO_WSTRING(readBuff[iIndex_2].sTxt_ENG);
							IF 16=iIndex_1 THEN
								EXIT;
							END_IF
						END_IF
					END_FOR
				1:
					FOR iIndex_2:=1 TO (MAX_IO_MODULE_NUM*16) BY 1 DO
						IF iCurrPage=readBuff[iIndex_2].nGroup AND iIndex_1=readBuff[iIndex_2].nNumber THEN
							HMIITF.sInfor[iIndex_1]:=readBuff[iIndex_2].sTxt_CHN;
							IF 16=iIndex_1 THEN
								EXIT;
							END_IF
						END_IF
					END_FOR
			END_CASE
		END_FOR
	END_IF
	bRefresh:=FALSE;
	
(*Read csv file*)
	IF NOT bInit THEN
		bInit:=TRUE;
		bReload:=TRUE;
	END_IF
	fbFileReadWrite(
		readBuff:= readBuff, 
		sFileName:= sFileName, 
		bRead:= bReload, 
		sTxtHead:= 'GROUP,NUM,ENG,CHN,NO USE', 
		bBusy=> , 
		bDone=> , 
		bError=> , 
		nErrid=> );
	IF bReload THEN
		bReload:=FALSE;
	END_IF
	Refresh_R_TRIG(CLK:=fbFileReadWrite.bDone);
	IF Refresh_R_TRIG.Q THEN
		bRefresh:=TRUE;
	END_IF

END_FUNCTION_BLOCK

// ---- POUs/BaseModule/IO/ReadWriteCSV/FB_IOFileReadWrite.TcPOU
FUNCTION_BLOCK FB_IOFileReadWrite
VAR_IN_OUT
	readBuff:ARRAY [*] OF ST_DataFmtBase;
END_VAR
VAR_INPUT
	sFileName:T_MaxString:='C:\CsvFilePath\csvfile.csv';//'Hard Disk\CsvFilePath\csvfile.csv'
	bRead:BOOL;
	sTxtHead:STRING:='GROUP,NUM,ENG,CHN,NO USE';
END_VAR
VAR_OUTPUT
	bBusy:BOOL;
	bDone:BOOL;
	bError:BOOL;
	nErrid:UDINT;
END_VAR
VAR
	fbFileOpen:FB_FileOpen;
	fbFileClose:FB_FileClose;
	fbFileGets:FB_FileGets;
	fbReader:FB_CSVMemBufferReader;
	hFile:UINT:= 0;
	
	sReadLine:STRING(255);
	bReadEOF:BOOL;
	nReadCount:DINT;
	
	nStepRead:UINT;
	nReadBuffMin:DINT;
	nReadBuffMax:DINT;
	nReadBuffLen:DINT;
END_VAR


nReadBuffMin:=LOWER_BOUND(readBuff,1);//获取不定长数组的最小下标
nReadBuffMax:=UPPER_BOUND(readBuff,1);//获取不定长数组的最大下标
nReadBuffLen:=nReadBuffMax-nReadBuffMin+1;//获取数组有效长度

readCSV();

//

METHOD PRIVATE createDir : BOOL
VAR
	sPathNameTemp	: T_MaxString := 'C:\TwinCAT\Data.txt';
	sDriveTemp		: STRING(3);
	sDirTemp		: T_MaxString;
	sFileNameTemp	: T_MaxString;
	sExtTemp		: T_MaxString;
	bSuccess		: BOOL;
	fbCreateDir		: FB_CreateDir;
	sFileDirTemp	: T_MaxString;
END_VAR
sPathNameTemp:=sFileName;
bSuccess := F_SplitPathName(sPathName:= sPathNameTemp,
						sDrive:= sDriveTemp,
						sDir:= sDirTemp,
						sFileName:= sFileNameTemp,
						sExt:= sExtTemp );
IF bSuccess THEN
	bSuccess:=FALSE;
	IF LEFT(sDirTemp,LEN(sDirTemp)-1)<>'' THEN
		sFileDirTemp:=CONCAT(STR1:=sDriveTemp,STR2:=LEFT(sDirTemp,LEN(sDirTemp)-1));
		fbCreateDir(
			sNetId:= , 
			sPathName:= sFileDirTemp, 
			ePath:= PATH_GENERIC, 
			bExecute:= TRUE, 
			tTimeout:= , 
			bBusy=> , 
			bError=> , 
			nErrId=> );
	END_IF
END_IF
fbCreateDir(
	sNetId:= , 
	sPathName:= , 
	ePath:= , 
	bExecute:= FALSE, 
	tTimeout:= , 
	bBusy=> , 
	bError=> , 
	nErrId=> );
END_METHOD

METHOD PRIVATE readCSV : BOOL
VAR_INPUT
END_VAR
VAR
	nTemp_readCSV:INT;
	sGetValue_temp:STRING(255);
	bRtn:BOOL;
	nTemp1:INT;
END_VAR
DEFAULT_CSV_FIELD_SEP:= 16#2C;  //配置CSV文件的分割符，16#2C表明各个参数之间是用逗号分隔的。

CASE nStepRead OF
	0:
		IF bRead THEN
			bRead:=FALSE;
			bBusy:=TRUE;
			bDone:=FALSE;
			bError:=FALSE;
			nErrid:=0;
			
			nReadCount:=nReadBuffMin;			
			MEMSET(readBuff,0,TO_UDINT(SIZEOF(readBuff[nReadCount])*nReadBuffLen));//清空内存
			nStepRead:=100;
		END_IF
	100:
		fbFileOpen(bExecute:=FALSE);
		nStepRead:=nStepRead+10;
	110:
		fbFileOpen(
			sNetId:= , 
			sPathName:= sFileName, 
			nMode:= FOPEN_MODEREAD OR FOPEN_MODETEXT, 
			ePath:= PATH_GENERIC, 
			bExecute:= TRUE, 
			tTimeout:= , 
			bBusy=> , 
			bError=> , 
			nErrId=> , 
			hFile=> hFile);
		IF NOT fbFileOpen.bBusy THEN
			IF NOT fbFileOpen.bError THEN
				nStepRead:=nStepRead+10;
			ELSE
				nErrid:=fbFileOpen.nErrId;
				nStepRead:=60000;//Error
			END_IF
		END_IF
	120:
		fbFileGets(bExecute:=FALSE);
		IF nReadCount>nReadBuffMax THEN
			nStepRead:=150;
		ELSE
			nStepRead:=nStepRead+10;
		END_IF
	130:
		fbFileGets(
			sNetId:= , 
			hFile:= hFile, 
			bExecute:= TRUE, 
			tTimeout:= , 
			bBusy=> , 
			bError=> , 
			nErrId=> , 
			sLine=> sReadLine, 
			bEOF=> bReadEOF);
		IF NOT fbFileGets.bBusy THEN
			IF NOT fbFileGets.bError THEN
				sReadLine:=CONCAT(STR1:=sReadLine,STR2:='$R$L');
				nStepRead:=nStepRead+10;
			ELSE
				nErrid:=fbFileGets.nErrId;
				nStepRead:=60000;//Error
			END_IF
		END_IF
	140:
		IF ''<>sTxtHead AND FIND(sReadLine,sTxtHead)>0 THEN
			nStepRead:=120;
			RETURN;
		END_IF
		nTemp1:=0;
		fbReader.eCmd:=eEnumCmd_First;(* Read first field value *)
		FOR nTemp_readCSV:=0 TO 3 DO
			fbReader(
				eCmd:= , 
				pBuffer:= ADR(sReadLine), 
				cbBuffer:= SIZEOF(sReadLine), 
				bOk=> , 
				getValue=> sGetValue_temp, 
				pValue=> , 
				cbValue=> , 
				bCRLF=> , 
				cbRead=> );
			IF fbReader.bOk THEN
				fbReader.eCmd:=eEnumCmd_Next;
				CASE nTemp_readCSV OF 
					0:
						readBuff[nReadCount].nGroup:=TO_DINT(sGetValue_temp);
					1:
						readBuff[nReadCount].nNumber:=TO_DINT(sGetValue_temp);
					2:
						readBuff[nReadCount].sTxt_ENG:=sGetValue_temp;
					3:
						bRtn:=UTF8_TO_WSTRING(ADR(readBuff[nReadCount].sTxt_CHN),ADR(sGetValue_temp),SIZEOF(sGetValue_temp));
						IF NOT bRtn OR ""=readBuff[nReadCount].sTxt_CHN THEN
							readBuff[nReadCount].sTxt_CHN:=TO_WSTRING(readBuff[nReadCount].sTxt_ENG);
						END_IF
				END_CASE
				nTemp1:=nTemp_readCSV;
			END_IF
		END_FOR
		IF NOT bReadEOF THEN
			nReadCount:=nReadCount+1;
			nStepRead:=120;
		ELSE
			nStepRead:=nStepRead+10;
		END_IF
	150:
		nStepRead:=50000;//Done

 //Done
	50000:
		fbFileOpen(bExecute:=FALSE);
		fbFileGets(bExecute:=FALSE);
		fbFileClose(bExecute:=FALSE);
		nStepRead:=nStepRead+10;
	50010:
		fbFileClose(
			sNetId:= , 
			hFile:= hFile, 
			bExecute:= TRUE, 
			tTimeout:= , 
			bBusy=> , 
			bError=> , 
			nErrId=> );
		IF NOT fbFileClose.bBusy THEN
			nStepRead:=nStepRead+10;
		END_IF
	50020:
		fbFileClose(bExecute:=FALSE);
		bBusy:=FALSE;
		bDone:=TRUE;
		bError:=FALSE;
		nStepRead:=0;
 //Error
	60000:
		fbFileOpen(bExecute:=FALSE);
		fbFileGets(bExecute:=FALSE);
		fbFileClose(bExecute:=FALSE);
		nStepRead:=nStepRead+10;
	60010:
		fbFileClose(
			sNetId:= , 
			hFile:= hFile, 
			bExecute:= TRUE, 
			tTimeout:= , 
			bBusy=> , 
			bError=> , 
			nErrId=> );
		IF NOT fbFileClose.bBusy THEN
			nStepRead:=nStepRead+10;
		END_IF
	60020:
		fbFileClose(bExecute:=FALSE);
		bBusy:=FALSE;
		bDone:=FALSE;
		bError:=TRUE;
		nStepRead:=0;
END_CASE
END_METHOD

END_FUNCTION_BLOCK

// ---- POUs/BaseModule/IO/FB_IOBase_Output_New.TcPOU
FUNCTION_BLOCK FB_IOBase_Output_New
VAR CONSTANT
	MAX_IO_MODULE_NUM:DINT:=15;
END_VAR
VAR_INPUT
	iIOModuleNum:DINT;//输入输出模块数量
	stIOBase:ARRAY [1..MAX_IO_MODULE_NUM] OF ST_OUTPUT_IO;
	iLanguage:UINT;//0：英文；1：中文
	sFileName:T_MaxString:='C:\IOFilePath\iocsvfile.csv';//'Hard Disk\IOFilePath\iocsvfile.csv'
	bReload:BOOL;//加载配置文件 触发
END_VAR
VAR_OUTPUT
END_VAR
VAR
	HMIITF:ST_IOBase_Show_HMI;
	
	iIOModuleNum_Temp:DINT;//输入输出模块数量
	
	next_R_TRIG:R_TRIG;
	back_R_TRIG:R_TRIG;
	targer_R_TRIG:R_TRIG;
	
	iCurrPage:DINT:=1;
	iIndex_1:DINT;
	iIndex_2:DINT;
	
	readBuff:ARRAY [1..MAX_IO_MODULE_NUM*16] OF ST_DataFmtBase;
	fbFileReadWrite:FB_IOFileReadWrite;
	bInit:BOOL;
	bRefresh:BOOL;
	Refresh_R_TRIG:R_TRIG;
	iLanguage_temp:UINT;//0：英文；1：中文
END_VAR


HMIITF.sIOType:='Output';

iIOModuleNum_Temp:=iIOModuleNum;
IF iIOModuleNum<0 THEN
	iIOModuleNum_Temp:=0;
ELSIF iIOModuleNum>MAX_IO_MODULE_NUM THEN
	iIOModuleNum_Temp:=MAX_IO_MODULE_NUM;
END_IF

(*HMI process*)
 (* Next button *)
	next_R_TRIG(CLK:=HMIITF.bNextPage);
	IF next_R_TRIG.Q THEN
		iCurrPage:=iCurrPage+1;
		bRefresh:=TRUE;
	END_IF
 (* Back button *)
	back_R_TRIG(CLK:=HMIITF.bBackPage);
	IF back_R_TRIG.Q THEN
		iCurrPage:=iCurrPage-1;
		bRefresh:=TRUE;
	END_IF
 (* Targer button *)
 	IF HMIITF.iTargerPage<=0 THEN
		HMIITF.iTargerPage:=iIOModuleNum_Temp;
	ELSIF HMIITF.iTargerPage>iIOModuleNum_Temp THEN
		HMIITF.iTargerPage:=1;
	END_IF
	targer_R_TRIG(CLK:=HMIITF.bTargerPage);
	IF targer_R_TRIG.Q THEN
		iCurrPage:=HMIITF.iTargerPage;
		bRefresh:=TRUE;
	END_IF

	IF iCurrPage<=0 THEN
		iCurrPage:=iIOModuleNum_Temp;
	ELSIF iCurrPage>iIOModuleNum_Temp THEN
		iCurrPage:=1;
	END_IF
	HMIITF.iCurrPage:=iCurrPage;
	HMIITF.iMaxPage:=iIOModuleNum_Temp;
	FOR iIndex_1:=1 TO 16 BY 1 DO
		HMIITF.bIO[iIndex_1]:=stIOBase[iCurrPage].io[iIndex_1];
	END_FOR
	IF bRefresh THEN
		FOR iIndex_1:=1 TO 16 BY 1 DO
			HMIITF.bIO[iIndex_1]:=stIOBase[iCurrPage].io[iIndex_1];
			
			CASE iLanguage_temp OF
				0:
					FOR iIndex_2:=1 TO (MAX_IO_MODULE_NUM*16) BY 1 DO
						IF iCurrPage=readBuff[iIndex_2].nGroup AND iIndex_1=readBuff[iIndex_2].nNumber THEN
							HMIITF.sInfor[iIndex_1]:=TO_WSTRING(readBuff[iIndex_2].sTxt_ENG);
							IF 16=iIndex_1 THEN
								EXIT;
							END_IF
						END_IF
					END_FOR
				1:
					FOR iIndex_2:=1 TO (MAX_IO_MODULE_NUM*16) BY 1 DO
						IF iCurrPage=readBuff[iIndex_2].nGroup AND iIndex_1=readBuff[iIndex_2].nNumber THEN
							HMIITF.sInfor[iIndex_1]:=readBuff[iIndex_2].sTxt_CHN;
							IF 16=iIndex_1 THEN
								EXIT;
							END_IF
						END_IF
					END_FOR
			END_CASE
		END_FOR
	END_IF
	bRefresh:=FALSE;
	
(*Read csv file*)
	IF NOT bInit THEN
		bInit:=TRUE;
		bReload:=TRUE;
	END_IF
	fbFileReadWrite(
		readBuff:= readBuff, 
		sFileName:= sFileName, 
		bRead:= bReload, 
		sTxtHead:= 'GROUP,NUM,ENG,CHN,NO USE', 
		bBusy=> , 
		bDone=> , 
		bError=> , 
		nErrid=> );
	IF bReload THEN
		bReload:=FALSE;
	END_IF
	Refresh_R_TRIG(CLK:=fbFileReadWrite.bDone);
	IF Refresh_R_TRIG.Q THEN
		bRefresh:=TRUE;
	END_IF
	IF iLanguage_temp<>iLanguage THEN
		iLanguage_temp:=iLanguage;
		bRefresh:=TRUE;
	END_IF

END_FUNCTION_BLOCK

// ---- POUs/BaseModule/SystemTimeModule/systemTimeModule.TcPOU
FUNCTION_BLOCK systemTimeModule (* 该功能块可提供系统时间; 可提供 *)
VAR_INPUT
END_VAR
VAR_OUTPUT
	systemTime		: TIMESTRUCT;
	timeInterval	: ARRAY [0..gSystemTimeMaxNum] OF UDINT;//  最大值为 gSystemTimeMaxNum		:UINT:=2000;
END_VAR
VAR
	//获取系统时间
	ntGetTime		: NT_GetTime;
	systemTimeTemp	: TIMESTRUCT;
	systemTimeStep	: UINT:=0;

	timeStartArray		: ARRAY [0..gSystemTimeMaxNum] OF TIME;//  最大值为 gSystemTimeMaxNum		:UINT:=2000;
	timeEndArray		: ARRAY [0..gSystemTimeMaxNum] OF TIME;//  最大值为 gSystemTimeMaxNum		:UINT:=2000;
	timeIntervalArray	: ARRAY [0..gSystemTimeMaxNum] OF TIME;//  最大值为 gSystemTimeMaxNum		:UINT:=2000;
	timeEnable			: ARRAY [0..gSystemTimeMaxNum] OF BOOL;//  最大值为 gSystemTimeMaxNum		:UINT:=2000;
END_VAR


(* 获取系统时间 *)
CASE systemTimeStep OF
0:
	ntGetTime(
		NETID:= , 
		START:= FALSE, 
		TMOUT:= , 
		BUSY=> , 
		ERR=> , 
		ERRID=> , 
		TIMESTR=> );
	IF NOT ntGetTime.BUSY AND NOT ntGetTime.ERR THEN
		systemTimeStep:=systemTimeStep+1;
	END_IF
1:
	ntGetTime(
		NETID:= , 
		START:= TRUE, 
		TMOUT:= , 
		BUSY=> , 
		ERR=> , 
		ERRID=> , 
		TIMESTR=> systemTimeTemp);
	IF NOT ntGetTime.BUSY AND NOT ntGetTime.ERR THEN
		systemTime:=systemTimeTemp;
	END_IF
	IF NOT ntGetTime.BUSY THEN
		systemTimeStep:=0;
	END_IF
END_CASE

(* 计算时间差 *)
METHOD calcTimeInterval : LREAL
VAR_INPUT
	timeStructBefore: TIMESTRUCT;//起始时间
	timeStructAfter: TIMESTRUCT;//结束时间
END_VAR
VAR
	timeStructTemp: TIMESTRUCT;
	timeBefor: DWORD;
	timeAfter: DWORD;
	dwordTimeInterval: DWORD;
	lrealTimeInterval: LREAL;
END_VAR
timeBefor:=(timeStructBefore.wYear*365*24*60*60*1000
					+timeStructBefore.wMonth*30*24*60*60*1000
					+timeStructBefore.wDay*24*60*60*1000
					+timeStructBefore.wHour*60*60*1000
					+timeStructBefore.wMinute*60*1000
					+timeStructBefore.wSecond*1000
					+timeStructBefore.wMilliseconds);
timeAfter:=(timeStructAfter.wYear*365*24*60*60*1000
					+timeStructAfter.wMonth*30*24*60*60*1000
					+timeStructAfter.wDay*24*60*60*1000
					+timeStructAfter.wHour*60*60*1000
					+timeStructAfter.wMinute*60*1000
					+timeStructAfter.wSecond*1000
					+timeStructAfter.wMilliseconds);

dwordTimeInterval:=ABS(timeAfter - timeBefor);
//lrealTimeInterval:=DWORD_TO_LREALEX(dwordTimeInterval)/1000;
lrealTimeInterval:=TO_LREAL(dwordTimeInterval)/1000.0;

calcTimeInterval:=lrealTimeInterval;
END_METHOD

(* 启用对应编号的计时器 *)
METHOD enableTime : BOOL
VAR_INPUT
	num		:UINT:=0;//时间计时编号  最大值为 gSystemTimeMaxNum		:UINT:=2000;
END_VAR
IF num >=gSystemTimeMaxNum THEN
	RETURN;
END_IF
timeEnable[num]:=TRUE;
enableTime:=timeEnable[num];
END_METHOD

(* 停止对应编号的计时器计时, 并返回开始时间到结束时间的时间间隔 *)
METHOD endTime : TIMESTRUCT
VAR_INPUT
	num		:UINT:=0;//时间计时编号  最大值为 gSystemTimeMaxNum		:UINT:=2000; 需要先执行timeEnable[num]:=TRUE;
END_VAR
IF num >=gSystemTimeMaxNum THEN
	RETURN;
END_IF
IF NOT timeEnable[num] THEN
	RETURN;
END_IF

timeEndArray[num]:=TIME();
endTime:=systemTime;

timeIntervalArray[num]:=timeEndArray[num]-timeStartArray[num];
timeInterval[num]:=TO_UDINT(timeIntervalArray[num]);
END_METHOD

(*系统时间，格式YYYY-MM-DD hh:mm:ss_zzz*)
METHOD getStrSysTime : STRING
VAR_INPUT
END_VAR
getStrSysTime:=SYSTEMTIME_TO_STRING(systemTime);//系统时间转成字符串格式
END_METHOD

(* 系统时间-日,格式xx *)
METHOD getStrSysTimeDD : STRING
VAR_INPUT
END_VAR
getStrSysTimeDD:=WORD_TO_DECSTR(in:=systemTime.wDay,iPrecision:=2);
END_METHOD

(* 系统时间-月,格式xx *)
METHOD getStrSysTimeMM : STRING
VAR_INPUT
END_VAR
getStrSysTimeMM:=WORD_TO_DECSTR(in:=systemTime.wMonth,iPrecision:=2);
END_METHOD

(* 系统时间-年,格式xxxx *)
METHOD getStrSysTimeYYYY : STRING
VAR_INPUT
END_VAR
getStrSysTimeYYYY:=WORD_TO_DECSTR(in:=systemTime.wYear,iPrecision:=4);
END_METHOD

(* 返回计时器编号的计时数值 UDINT类型 ms单位 *)
METHOD getTimeInterval : UDINT
VAR_INPUT
	num		:UINT:=0;//时间计时编号  最大值为 gSystemTimeMaxNum		:UINT:=2000; 需要先执行timeEnable[num]:=TRUE;
END_VAR
IF num >=gSystemTimeMaxNum THEN
	RETURN;
END_IF
IF NOT timeEnable[num] THEN
	RETURN;
END_IF

getTimeInterval:=timeInterval[num];
END_METHOD

(* 返回计时器编号的计时数值 STRING 类型 *)
METHOD getTimeIntervalStr : STRING(255)
VAR_INPUT
	num				:UINT:=0;//时间计时编号  最大值为 gSystemTimeMaxNum		:UINT:=2000; 需要先执行timeEnable[num]:=TRUE;
	prefixStr		:STRING(255):='';//打印时间间隔 添加的前缀字符串
	suffixStr		:STRING(255):='';//打印时间间隔 添加的后缀字符串
END_VAR
VAR
	sTemp			:STRING(255):='';
	sTimeTemp		:STRING(255):='';
END_VAR
IF num >=gSystemTimeMaxNum THEN
	RETURN;
END_IF
IF NOT timeEnable[num] THEN
	RETURN;
END_IF

sTimeTemp:=TO_STRING(timeIntervalArray[num]);
sTimeTemp:=DELETE(sTimeTemp,2,1);

sTemp:=prefixStr;
sTemp:=CONCAT(sTemp,sTimeTemp);
sTemp:=CONCAT(sTemp,suffixStr);

getTimeIntervalStr:=sTemp;
END_METHOD

(* 启动对应编号的计时器计时, 并返回开始时间到结束时间的时间间隔 *)
METHOD startTime : TIMESTRUCT
VAR_INPUT
	num		:UINT:=0;//时间计时编号  最大值为 gSystemTimeMaxNum		:UINT:=2000; 需要先执行timeEnable[num]:=TRUE;
END_VAR
IF num >=gSystemTimeMaxNum THEN
	RETURN;
END_IF
IF NOT timeEnable[num] THEN
	RETURN;
END_IF

timeStartArray[num]:=TIME();
startTime:=systemTime;
END_METHOD

ACTION VersionLog:
(*
版本: V1.0.0.0
说明:
	1. 首个版本
(**************************************************)
*)
END_ACTION

END_FUNCTION_BLOCK

// ---- POUs/Other/MachineState/FB_MachineState.TcPOU
FUNCTION_BLOCK FB_MachineState
VAR_INPUT
	RunningState			:RunningStatus:=RunningStatus.eManualState;// 整机设备的运行状态
	HMI_E_Stop				:BOOL:=TRUE;// HMI E-Stop 按钮
	HMI_Start				:BOOL:=FALSE;// HMI Start 按钮
	HMI_Stop				:BOOL:=FALSE;// HMI Stop 按钮
	HMI_Reset				:BOOL:=FALSE;// HMI Reset 按钮
	HMI_EnableBuzzer		:BOOL:=FALSE;// HMI 启用蜂鸣器
	HMI_AllStop				:BOOL;
	HMI_Version				:STRING:='V1.0.0';
	Actual_E_Stop			:BOOL:=TRUE;// 设备 E-Stop 按钮
	Actual_Start			:BOOL;// 设备 Start 按钮
	Actual_Stop				:BOOL;// 设备 Stop 按钮
	Actual_Reset			:BOOL;// 设备 Reset 按钮
	iLanguage				:UINT;// 0：英文；1：中文
END_VAR
VAR_OUTPUT
	E_Stop					:BOOL:=TRUE;
	Reset					:BOOL:=FALSE;
	Stop					:BOOL:=FALSE;
	Start					:BOOL:=FALSE;
	StartLamp				:BOOL:=FALSE;// Start 按钮灯
	StopLamp				:BOOL:=FALSE;// Stop 按钮灯
	ResetLamp				:BOOL:=FALSE;// Reset 按钮灯
	// 三色灯
	RedLamp					:BOOL:=FALSE;// red 按钮灯
	GreenLamp				:BOOL:=FALSE;// Green 按钮灯
	YellowLamp				:BOOL:=FALSE;// Yellow 按钮灯
	Buzzer					:BOOL:=FALSE;// Buzzer
	AllStop					:BOOL;// 只保持一个周期TRUE
	RunStateTxt				:WSTRING:="";// HMI 运行状态文本显示
	RunStateTxtS			:WSTRING:="";// HMI 运行状态文本显示 单个字母
END_VAR
VAR
	pauseStateTON1			:TON;
	pauseStateTON2			:TON;
	stopStateTON1			:TON;
	stopStateTON2			:TON;
	errorStateTON1			:TON;
	errorStateTON2			:TON;
	homeStateTON1			:TON;
	homeStateTON2			:TON;
	allStop_R_TRIG			:R_TRIG;
END_VAR

(* 按钮、三色灯 *)
	E_Stop:=HMI_E_Stop OR Actual_E_Stop;//后续需要改回AND
	Start:=HMI_Start OR Actual_Start;
	Stop:=HMI_Stop OR Actual_Stop;
	Reset:=HMI_Reset OR Actual_Reset;
	AllStop:=FALSE;
	allStop_R_TRIG(CLK:=HMI_AllStop);
	IF allStop_R_TRIG.Q THEN
		AllStop:=TRUE;
	END_IF
(* 状态监控 *)
	CASE RunningState OF
		RunningStatus.eManualState:
			IF 1=iLanguage THEN // 中文
				RunStateTxt:="手动运行中";
			ELSE
				RunStateTxt:="Manual running";
			END_IF
			RunStateTxtS:="M";
			// StartLamp:=FALSE;
			StopLamp:=FALSE;
			// ResetLamp:=FALSE;
			RedLamp:=FALSE;
			GreenLamp:=FALSE;
			// YellowLamp:=FALSE;
			Buzzer:=FALSE;
				
			StartLamp:=TRUE;
			ResetLamp:=TRUE;
			YellowLamp:=TRUE;
		RunningStatus.eAutoState:
			IF 1=iLanguage THEN // 中文
				RunStateTxt:="自动运行中";
			ELSE
				RunStateTxt:="Auto running";
			END_IF
			RunStateTxtS:="A";
			StartLamp:=FALSE;
			// StopLamp:=FALSE;
			ResetLamp:=FALSE;
			RedLamp:=FALSE;
			// GreenLamp:=FALSE;
			YellowLamp:=FALSE;
			Buzzer:=FALSE;
			
			StopLamp:=TRUE;
			GreenLamp:=TRUE;
		RunningStatus.ePauseState:
			IF 1=iLanguage THEN // 中文
				RunStateTxt:="暂停运行中";
			ELSE
				RunStateTxt:="Pause running";
			END_IF
			RunStateTxtS:="P";
			// StartLamp:=FALSE;
			// StopLamp:=FALSE;
			ResetLamp:=FALSE;
			RedLamp:=FALSE;
			// GreenLamp:=FALSE;
			YellowLamp:=FALSE;
			Buzzer:=FALSE;
				
			StopLamp:=TRUE;
			pauseStateTON1(IN:=NOT GreenLamp, PT:=T#0.5S);
			pauseStateTON2(IN:=GreenLamp, PT:=T#0.5S);
			IF pauseStateTON1.Q THEN
				StartLamp:=TRUE;
				GreenLamp:=TRUE;
			END_IF
			IF pauseStateTON2.Q THEN
				StartLamp:=FALSE;
				GreenLamp:=FALSE;
			END_IF
		RunningStatus.eStopState:
			IF 1=iLanguage THEN // 中文
				RunStateTxt:="停止运行中";
			ELSE
				RunStateTxt:="Stop running";
			END_IF
			RunStateTxtS:="S";
			StartLamp:=FALSE;
			StopLamp:=FALSE;
			ResetLamp:=FALSE;
			RedLamp:=FALSE;
			// GreenLamp:=FALSE;
			// YellowLamp:=FALSE;
			Buzzer:=FALSE;
				
			GreenLamp:=TRUE;
			stopStateTON1(IN:=NOT YellowLamp, PT:=T#0.5S);
			stopStateTON2(IN:=YellowLamp, PT:=T#0.5S);
			IF stopStateTON1.Q THEN
				YellowLamp:=TRUE;
			END_IF
			IF stopStateTON2.Q THEN
				YellowLamp:=FALSE;
			END_IF
		RunningStatus.eErrorState:
			IF 1=iLanguage THEN // 中文
				RunStateTxt:="报错运行中";
			ELSE
				RunStateTxt:="Error running";
			END_IF
			RunStateTxtS:="E";
			StartLamp:=FALSE;
			StopLamp:=FALSE;
			// ResetLamp:=FALSE;
			// RedLamp:=FALSE;
			GreenLamp:=FALSE;
			YellowLamp:=FALSE;
			// Buzzer:=FALSE;
				
			RedLamp:=TRUE;
			errorStateTON1(IN:=NOT ResetLamp, PT:=T#0.5S);
			errorStateTON2(IN:=ResetLamp, PT:=T#0.5S);
			IF errorStateTON1.Q THEN
				ResetLamp:=TRUE;
				Buzzer:=TRUE;
			END_IF
			IF errorStateTON2.Q THEN
				ResetLamp:=FALSE;
				Buzzer:=FALSE;
			END_IF
		RunningStatus.eHomeState:
			IF 1=iLanguage THEN // 中文
				RunStateTxt:="回原点运行中";
			ELSE
				RunStateTxt:="Home running";
			END_IF
			RunStateTxtS:="H";
			StartLamp:=FALSE;
			StopLamp:=FALSE;
			ResetLamp:=FALSE;
			RedLamp:=FALSE;
			GreenLamp:=FALSE;
			// YellowLamp:=FALSE;
			Buzzer:=FALSE;
			
			homeStateTON1(IN:=NOT YellowLamp, PT:=T#0.5S);
			homeStateTON2(IN:=YellowLamp, PT:=T#0.5S);
			IF homeStateTON1.Q THEN
				YellowLamp:=TRUE;
			END_IF
			IF homeStateTON2.Q THEN
				YellowLamp:=FALSE;
			END_IF
	END_CASE
IF NOT HMI_EnableBuzzer THEN
	Buzzer:=FALSE;
END_IF

END_FUNCTION_BLOCK

// ---- POUs/BaseModule/ActionModule/HEATModule/HeatModule.TcPOU
(*
--报错编号0: 无报错
--报错编号1: Heatting Error
*)
FUNCTION_BLOCK HeatModule
VAR_IN_OUT
	WarmHMI					:WARMStruct;
END_VAR
VAR_INPUT
	HeatType					:HeatType:=HEATType_Default;//设置加热器的类型, 可通过该变量修改为其他类型加热器
	
	real_TimeMonitor			:BOOL:=TRUE;//实时状态检测
	
	heat						:BOOL:=FALSE;// 加热触发信号
	ATLearning					:BOOL:=FALSE;// 加热自学习触发信号
	MVManul						:BOOL:=FALSE;// 手动控制
	heatCondition				:BOOL:=TRUE;// 加热启停条件
	ATLCondition				:BOOL:=TRUE;// 自学习启停条件
	MVCondition					:BOOL:=TRUE;// 手动控制启停条件
	reset						:BOOL:=FALSE;// 复位信号
	stop						:BOOL:=FALSE;// 停止信号
	power						:BOOL:=TRUE;// 加热动作后是否关闭继电器得电状态, TRUE--保持得电,FALSE--断开得电
	enable						:BOOL:=TRUE;// 加热禁用条件
	//ctrlMode					:ControlMode:=ControlMode.eManualCtrMode;//eManualCtrMode or eAutoCtrMode
	hmiEN						:BOOL:=TRUE;//HMI 启用条件
	
	errorID						:UDINT:=0;//加热错误报警分配的起始ID
	nameTXT						:STRING(255):='';//加热名字
	
	ctrl_heatStart				: BOOL;//bit0 开始加热
	
	para_SV						:REAL;// 温度设定值
	para_HLimit					:REAL:=200.0;// 温控报警上限参数
	para_LLimit					:REAL:=-10.0;// 温控报警下限参数
	para_setTOffset				:REAL:=1.0;// 温控偏差值
	HMIItf						:HEATModuleHMI;//每个加热对象都关联了一个HMI
	noteWTXT					:WSTRING(255):="";//气缸动作NoteTXT 中文
END_VAR
VAR_OUTPUT
	status_PV					:REAL;// 温控反馈测量值
	status_MV					:INT;// 温控反馈Manul设定值
	status_OutAndAlm			:INT;// 温控反馈输出状态及报警信息
	status_P					:INT;// 温控反馈P参数
	status_I					:INT;// 温控反馈I参数
	status_D					:INT;// 温控反馈D参数
		
	//heatRelay					:BOOL;// 加热输出
	note_heat					:BOOL:=false;// 加热触发无法执行
	busy						:BOOL;//加热动作Busy状态
	done						:BOOL;//加热动作Done状态
	heatdone					:BOOL;//加热动作完成
	ATLdone						:BOOL;// AT加热动作完成
	manuldone					:BOOL;// Manul加热动作完成
	error						:BOOL;//加热动作error状态
	errID						:UDINT;//加热动作errID
	errTXT						:STRING(255):='';//加热动作errTXT
	errWTXT						:WSTRING(255):="";//加热动作errTXT 中文
	heatting					:BOOL;// 加热中标志位
	status_OperSta				:UINT;// 温控反馈运行状态
END_VAR
	
VAR
		
	errorDelayTime				:TIME:=T#3000MS;//加热感应器感应超时
	//doneDelayTimeShort			:TIME:=T#100MS;//加热感应到位延时---取消使用
	//doneDelayTimeLong			:TIME:=T#500MS;//无加热感应到位延时---取消使用
	doneDelayTimeShortHeat		:TIME:=T#100MS;//加热感应到位延时_
	doneDelayTimeLongHeat		:TIME:=T#500MS;//无加热感应到位延时_
	
	ctrl_heatATStart			: BOOL;//bit2 100%AT实行中
	ctrl_heatATStop				: BOOL;//bit4 AT取消
	ctrl_heatAuto				: BOOL;//bit5 0: Auto,1: Manul
	ctrl_OperCmd				: UINT;// 控制命令字

	para_Manual_MV				:INT;// 手动MV	
	//para_OperCmd				:INT;// 命令字，链接加热ECT数据
	para_P						:INT;// 温控P参数
	para_I						:INT;// 温控I参数
	para_D						:INT;// 温控D参数
	
	Set_SV						AT%Q* :INT;// 温度设定值
	Set_Manual_MV				AT%Q* :INT;// 手动MV	
	Set_OperCmd					AT%Q* :UINT;// 命令字，链接加热ECT数据
	Set_P						AT%Q* :INT;// 温控P参数
	Set_I						AT%Q* :INT;// 温控I参数
	Set_D						AT%Q* :INT;// 温控D参数
		
	heatErrorDelayTon			:Ton;
	heatDoneDelayTon			:Ton;
	
	heatTrigRAlc				:R_Trig;//上升沿触发
	
	heatTrigR1					:R_Trig;//上升沿触发
	heatTrigR1_Aiko				:R_Trig;//上升沿触发
	manuleTrigR1				:R_Trig;//上升沿触发
	ATLTrigR1					:R_Trig;//上升沿触发
	resetTrigR1					:R_Trig;//上升沿触发
	stopTrigR1					:R_Trig;//上升沿触发
	powerTrigR1					:R_Trig;//上升沿触发
	
	heatStep					:UINT:=0;
	atlStep						:UINT:=0;
	manulStep					:UINT:=0;
	errorStep					:UINT:=0;
	
	notBusyMonitorDelayTon		:TON;//动作不切换时，延迟检测
	notBusyMonitorDelayTime 	:TIME:=T#2S;//动作不切换延迟检测时间
	firstPower			   		:BOOL:=FALSE;//首次上电标志位
	
	ATLearRest					:TON;// AT Learning 参数自复位
	
	HeatDoneTon					:TON; // 加热完成检测超时时间
	
	Act_PV					AT%I* :INT;// 温控反馈测量值
	Act_MV					AT%I* :INT;// 温控反馈Manul设定值
	Act_OutAndAlm			AT%I* :INT;// 温控反馈输出状态及报警信息
	Act_P					AT%I* :INT;// 温控反馈P参数
	Act_I					AT%I* :INT;// 温控反馈I参数
	Act_D					AT%I* :INT;// 温控反馈D参数
	Act_OperSta					AT%I* :UINT;// 温控反馈运行状态
END_VAR

Init_ACT();
Error_ACT();
Heat_ACT();
ATL_ACT();
Manul_ACT();
Reset_ACT();
Error_ACT();
SafeMonitor_ACT();
IOMap();

(*
触发伸出动作，成功触发返回TRUE，触发失败返回FALSE
*)
METHOD Act_ATL : BOOL
VAR_INPUT
	;
END_VAR
IF enable AND ATLearning THEN// AND NOT busy
	Act_ATL:=ATLearning:=TRUE;
ELSE
	Act_ATL:=FALSE;
END_IF
END_METHOD

(*
触发伸出动作，成功触发返回TRUE，触发失败返回FALSE
*)
METHOD Act_Heat : BOOL
VAR_INPUT
	//heatSV:INT;
END_VAR
IF enable AND heatCondition THEN// AND NOT busy
	Act_Heat:=heat:=TRUE;
	//para_SV:=heatSV;
ELSE
	Act_Heat:=FALSE;
END_IF
END_METHOD

(*
触发复位报警动作，成功触发返回TRUE，触发失败返回FALSE
*)
METHOD Act_Reset : BOOL
VAR_INPUT
END_VAR
Act_Reset:=reset:=TRUE;
END_METHOD

(*
触发停止输出动作，成功触发返回TRUE，触发失败返回FALSE
*)
METHOD Act_Stop : BOOL
VAR_INPUT
END_VAR
Act_Stop:=stop:=TRUE;
END_METHOD

ACTION ATL_ACT:
//自学习控制输出
IF ATLearning AND enable AND ATLCondition AND NOT busy THEN// AND NOT busy
	busy:=TRUE;
	ATLdone:=FALSE;
	heatdone:=FALSE;
	manuldone:=FALSE;
	atlStep:=10;
	note_heat:=FALSE;
	//errorStep:=0;
END_IF
ATLearning:=FALSE;

CASE atlStep OF
0:
	//ready
	
10:
	heatErrorDelayTon(IN:=FALSE);
	heatDoneDelayTon(IN:=FALSE);
	
	IF para_SV<para_HLimit AND para_SV>para_LLimit THEN//温度设定正常
		atlStep:=11;
	ELSE
		errorStep:=1;//加热设置错误
		atlStep:=60;
	END_IF
11:
	IF NOT status_OperSta.0 THEN// 非自动运行中
		atlStep:=13;
	ELSE
		errorStep:=5;
		atlStep:=60;
	END_IF
13:
	ctrl_OperCmd.2:=1;// AT 执行
	atlStep:=20;
	
20:
	heatErrorDelayTon(IN:=(NOT status_OperSta.2),PT:=errorDelayTime);
	IF heatErrorDelayTon.Q THEN
		//done:=FALSE;
		ATLdone:=FALSE;
		errorStep:=6;// 等待AT加热反馈超时
		RETURN;
	END_IF
	heatDoneDelayTon(IN:=status_OperSta.2,PT:=doneDelayTimeShortHeat);
	
	IF heatDoneDelayTon.Q THEN
		errorStep:=0;
		atlStep:=30;
		heatErrorDelayTon(IN:=FALSE);
		heatDoneDelayTon(IN:=FALSE);
	END_IF
30:
	IF NOT status_OperSta.2 THEN//等待AT完成
		errorStep:=0;
		atlStep:=50;
		heatErrorDelayTon(IN:=FALSE);
		heatDoneDelayTon(IN:=FALSE);
	END_IF
	IF status_OutAndAlm.0 OR status_OutAndAlm.1 OR status_OutAndAlm.2 OR status_OutAndAlm.3
	OR status_OutAndAlm.4 OR status_OutAndAlm.5 OR status_OutAndAlm.6 THEN
		errorStep:=3;
		heatStep:=60;
	END_IF
50:
	busy:=FALSE;
	ATLdone:=TRUE;
60://报错
	ctrl_OperCmd.0:=0;
	ctrl_OperCmd.4:=1;// AT 取消执行
	busy:=FALSE;
	ATLdone:=FALSE;
END_CASE
END_ACTION

ACTION Error_ACT:
CASE errorStep OF
	0:
		error:=FALSE;
		errID:=0;
		errTXT:='';
 (*
	1:
		error:=TRUE;
		errID:=errorID+errorStep;
		errTXT:=CONCAT(STR1:=nameTXT,STR2:=' Extend Error!');
		errWTXT:=WCONCAT(STR1:=TO_WSTRING(nameTXT),STR2:=" 伸出(打开)错误");
	2:
		error:=TRUE;
		errID:=errorID+errorStep;
		errTXT:=CONCAT(STR1:=nameTXT,STR2:=' Retract Error!');
		errWTXT:=WCONCAT(STR1:=TO_WSTRING(nameTXT),STR2:=" 缩回(关闭)错误");
		*)
	1..8:
		error:=TRUE;
		errID:=getErrID(errorStep);
		errTXT:=getErrTXT(errorStep);
		errWTXT:=getErrWTXT(errorStep);
END_CASE
END_ACTION

METHOD Get_Done_Heat : BOOL
VAR_INPUT
END_VAR
Get_Done_Heat:=heatdone;
END_METHOD

METHOD getErrID : UDINT
VAR_INPUT
	errID					:UDINT;//取值范围1~2
END_VAR
VAR
	nErrID					:UDINT;
END_VAR
nErrID:=errorID+errID;

getErrID:=nErrID;
END_METHOD

METHOD getErrTXT : STRING(255)
VAR_INPUT
	errID					:UDINT;//取值范围1~2
END_VAR
VAR
	sErrTXT					:STRING(255);
END_VAR

CASE errID OF
	1:
		sErrTXT:=CONCAT(STR1:=nameTXT,STR2:=' heat Error!');
	2:
		sErrTXT:=CONCAT(STR1:=nameTXT,STR2:=' stopheat Error!');
	3:
		sErrTXT:=CONCAT(STR1:=nameTXT,STR2:=' heat Return Statues Error!');
	4:
		sErrTXT:=CONCAT(STR1:=nameTXT,STR2:=' ATing Heat Error!');
	5:
		sErrTXT:=CONCAT(STR1:=nameTXT,STR2:=' Manuling Heat Error!');
	6:
		sErrTXT:=CONCAT(STR1:=nameTXT,STR2:=' AT Heat TimeOUT Error!');
	7:
		sErrTXT:=CONCAT(STR1:=nameTXT,STR2:=' Manule Heat Control Error!');
	8:
		sErrTXT:=CONCAT(STR1:=nameTXT,STR2:=' Heat TimeOut Error!');
ELSE
	sErrTXT:=CONCAT(STR1:=nameTXT,STR2:='');
END_CASE
getErrTXT:=sErrTXT;
END_METHOD

METHOD getErrWTXT : WSTRING(255)
VAR_INPUT
	errID					:UDINT;//取值范围1~16
END_VAR
VAR
	sErrTXT					:WSTRING(255);
END_VAR

CASE errID OF
	1:
		sErrTXT:=WCONCAT(STR1:=TO_WSTRING(nameTXT),STR2:=" 启动加热错误");
	2:
		sErrTXT:=WCONCAT(STR1:=TO_WSTRING(nameTXT),STR2:=" 停止加热错误");
	3:
		sErrTXT:=WCONCAT(STR1:=TO_WSTRING(nameTXT),STR2:=" 加热反馈异常");
	4:
		sErrTXT:=WCONCAT(STR1:=TO_WSTRING(nameTXT),STR2:=" AT中加热异常");
	5:
		sErrTXT:=WCONCAT(STR1:=TO_WSTRING(nameTXT),STR2:=" 手动中自动加热异常");
	6:
		sErrTXT:=WCONCAT(STR1:=TO_WSTRING(nameTXT),STR2:=" 等待AT执行超时");
	7:
		sErrTXT:=WCONCAT(STR1:=TO_WSTRING(nameTXT),STR2:=" 手动控制失控");
	8:
		sErrTXT:=WCONCAT(STR1:=TO_WSTRING(nameTXT),STR2:=" 加热超时");
ELSE
	sErrTXT:=WCONCAT(STR1:=TO_WSTRING(nameTXT),STR2:="");
END_CASE
getErrWTXT:=sErrTXT;
END_METHOD

ACTION Heat_ACT:
//正常加热控制输出
IF heat AND NOT heatCondition THEN
	note_heat:=FALSE;
END_IF
IF heat AND enable AND heatCondition AND NOT status_OperSta.2 AND NOT busy THEN// AND NOT busy
	busy:=TRUE;
	ATLdone:=FALSE;
	heatdone:=FALSE;
	manuldone:=FALSE;
	heatStep:=10;
	heatting:=FALSE;
	note_heat:=FALSE;
	//errorStep:=0;
END_IF
heat:=FALSE;

CASE heatStep OF
0:
	//ready
	
10:
	heatErrorDelayTon(IN:=FALSE);
	heatDoneDelayTon(IN:=FALSE);
	HeatDoneTon(IN:=FALSE);
	IF para_SV<para_HLimit AND para_SV>para_LLimit THEN//温度设定正常
		heatStep:=11;
	ELSE
		errorStep:=1;//加热设置错误
		heatStep:=60;
	END_IF
11:
	IF NOT status_OperSta.2 THEN// 非AT中
		heatStep:=12;
	ELSE
		errorStep:=4;
		heatStep:=60;
	END_IF
12:
	ctrl_heatStart:=TRUE;
	status_OperSta.5:=0;
	heatStep:=13;
13:
	ctrl_OperCmd.0:=ctrl_heatStart;
	heatStep:=20;
	
20:
	IF NOT( para_SV<para_HLimit AND para_SV>para_LLimit) THEN//温度设定正常
		errorStep:=1;//加热设置错误
		heatStep:=60;
		RETURN;
	END_IF
	heatErrorDelayTon(IN:=(NOT status_OperSta.0),PT:=errorDelayTime);
	IF heatErrorDelayTon.Q THEN
		//done:=FALSE;
		heatdone:=FALSE;
		errorStep:=1;// 等待加热反馈超时
		heatStep:=60;
		heatErrorDelayTon(IN:=FALSE);
		RETURN;
	END_IF
	heatDoneDelayTon(IN:=status_OperSta.0,PT:=doneDelayTimeShortHeat);
	
	IF heatDoneDelayTon.Q THEN
		IF status_OperSta.0 THEN
			errorStep:=0;
			heatStep:=30;
			heatting:=TRUE;
			heatErrorDelayTon(IN:=FALSE);
			heatDoneDelayTon(IN:=FALSE);
		ELSE
			IF status_OperSta.2 THEN//AT 中，报错
				busy:=FALSE;
				heatdone:=FALSE;
				errorStep:=3;
				heatStep:=60;
				heatErrorDelayTon(IN:=FALSE);
				heatDoneDelayTon(IN:=FALSE);
			END_IF
		END_IF
	END_IF
30:
	HeatDoneTon(IN:=ABS(para_SV-status_PV)>=para_setTOffset,PT:=DINT_TO_TIME(HMIItf.heatDoneCheckMaxTime*1000));
	IF HeatDoneTon.Q THEN
		errorStep:=8;
		heatStep:=60;
		HeatDoneTon(IN:=FALSE);
		RETURN;
	END_IF
	IF ABS(para_SV-status_PV)<para_setTOffset-0.1 THEN
		errorStep:=0;
		heatStep:=50;
		heatErrorDelayTon(IN:=FALSE);
		heatDoneDelayTon(IN:=FALSE);
	END_IF
	IF status_OutAndAlm.0 OR status_OutAndAlm.1 OR status_OutAndAlm.2 OR status_OutAndAlm.3
	OR status_OutAndAlm.4 OR status_OutAndAlm.5 OR status_OutAndAlm.6 THEN
		errorStep:=3;
		heatStep:=60;
	END_IF
50:
	busy:=FALSE;
	heatdone:=TRUE;
	heatting:=FALSE;
	IF ABS(para_SV-status_PV)>para_setTOffset THEN
		heatErrorDelayTon(IN:=FALSE);
		heatDoneDelayTon(IN:=FALSE);
		HeatDoneTon(IN:=FALSE);
		busy:=TRUE;
		heatdone:=FALSE;
		heatStep:=20;//重新返回检测
	END_IF
60://报错

	ctrl_heatStart:=FALSE;
	ctrl_OperCmd.0:=ctrl_heatStart;
	busy:=FALSE;
	heatdone:=FALSE;
END_CASE
END_ACTION

ACTION Init_ACT:
IF status_OutAndAlm.0 OR status_OutAndAlm.1 OR status_OutAndAlm.2 OR status_OutAndAlm.3
OR status_OutAndAlm.4 OR status_OutAndAlm.5 OR status_OutAndAlm.6 OR
NOT( status_PV<para_HLimit AND status_PV>para_LLimit) THEN
	stop:=TRUE;
	ctrl_heatStart:=FALSE;
	ctrl_OperCmd.0:=ctrl_heatStart;
END_IF
done:=(heatdone OR manuldone OR ATLdone);
InitHMI_ACT();
manualCtrl_ACT();
END_ACTION

ACTION InitHMI_ACT:
HMIItf.done:=done;
HMIItf.busy:=busy;
HMIItf.error:=error;
HMIItf.errID:=UDINT_TO_DINT(errID);
HMIItf.errTXT:=errTXT;
HMIItf.power:=power;
HMIItf.nameTXT:=nameTXT;

HMIItf.status_PV:=status_PV;// 温控反馈测量值
HMIItf.status_MV:=status_MV;// 温控反馈Manul设定值
HMIItf.oheatStart:=busy AND ctrl_OperCmd.0;// 加热在执行
HMIItf.iheatStart:=heatting AND status_OperSta.0 AND ctrl_OperCmd.0; // 加热运行中
HMIItf.status_P:=Act_P;// 温控反馈P参数
HMIItf.status_I:=Act_I;// 温控反馈I参数
HMIItf.status_D:=Act_D;// 温控反馈D参数

//para_HLimit:=HMIItf.para_HLimit;// 温控最大值
para_SV:=HMIItf.para_SV;// 温度设定值
para_Manual_MV:=HMIItf.para_Manual_MV;
para_setTOffset:=HMIItf.para_setTOffset;
END_ACTION

ACTION IOMap:
status_PV:=INT_TO_REAL(Act_PV)*0.1;
status_OutAndAlm:=Act_OutAndAlm;
status_MV:=Act_MV;
status_OperSta:=Act_OperSta;



Set_OperCmd:=ctrl_OperCmd;
Set_SV:=REAL_TO_INT(para_SV)*10;
Set_Manual_MV:=para_Manual_MV;
END_ACTION

ACTION ManualCtrl_ACT:
//HMI手动控制
//IF ctrlMode=eManualCtrMode THEN
IF hmiEN THEN
//	extendTrigRAlc(CLK:=HMIItf.extendAndretract);
//	IF extendTrigRAlc.Q THEN// AND NOT busy
//		IF extRelay THEN//如果伸出继电器或伸出传感器亮，则认为已经伸出过
//			retract:=TRUE;
//		END_IF
//		IF retRelay THEN
//			extend:=TRUE;
//		END_IF
//		IF NOT extRelay AND NOT retRelay THEN
//			IF extAprSw THEN
//				retract:=TRUE;
//			END_IF
//			IF retAprSw THEN
//				extend:=TRUE;
//			END_IF
//		END_IF
//	END_IF
	heatTrigR1_Aiko(CLK:=HMIItf.bHeat);
	IF heatTrigR1_Aiko.Q AND NOT ctrl_heatStart AND NOT status_OperSta.0 THEN// AND NOT busy
		para_SV:=HMIItf.para_SV;
		heat:=TRUE;
	END_IF
	IF heatTrigR1_Aiko.Q AND (ctrl_heatStart OR status_OperSta.0) THEN// AND NOT busy
		para_SV:=0;
		para_Manual_MV:=0;
		stop:=TRUE;
	END_IF
	heatTrigR1(CLK:=HMIItf.heat);
	IF heatTrigR1.Q THEN// AND NOT busy
		para_SV:=HMIItf.para_SV;
		heat:=TRUE;
	END_IF
	ATLTrigR1(CLK:=HMIItf.ATLearning);
	IF ATLTrigR1.Q THEN// AND NOT busy
		para_SV:=HMIItf.para_SV;
		ATLearning:=TRUE;
	END_IF
	manuleTrigR1(CLK:=HMIItf.manuleHeat);
	IF manuleTrigR1.Q THEN// AND NOT busy
		para_Manual_MV:=HMIItf.para_Manual_MV;
		MVManul:=TRUE;
	END_IF
		
	resetTrigR1(CLK:=HMIItf.reset);
	IF resetTrigR1.Q THEN// AND NOT busy
		para_SV:=0;
		para_Manual_MV:=0;
		reset:=TRUE;
	END_IF
	
	stopTrigR1(CLK:=HMIItf.stop);
	IF stopTrigR1.Q THEN// AND NOT busy
		para_SV:=0;
		para_Manual_MV:=0;
		stop:=TRUE;
	END_IF
	powerTrigR1(CLK:=HMIItf.power);
	IF powerTrigR1.Q THEN// AND NOT busy
		IF power THEN
			power:=FALSE;
		ELSE
			power:=TRUE;
		END_IF
	END_IF
END_IF
END_ACTION

ACTION Manul_ACT:
//手动加热比例设置输出
IF MVManul AND enable AND MVCondition AND NOT busy THEN// AND NOT busy
	busy:=TRUE;
	ATLdone:=FALSE;
	heatdone:=FALSE;
	manuldone:=FALSE;
	manulStep:=10;
	note_heat:=FALSE;
	//errorStep:=0;
END_IF
MVManul:=FALSE;

CASE manulStep OF
0:
	//ready
	
10:
	heatErrorDelayTon(IN:=FALSE);
	heatDoneDelayTon(IN:=FALSE);
	
	IF para_Manual_MV<30 AND para_Manual_MV>0.1 THEN//温度设定正常
		manulStep:=11;
	ELSE
		errorStep:=1;//加热设置错误
		manulStep:=60;
	END_IF
11:
	IF NOT status_OperSta.0 AND NOT status_OperSta.2 THEN// 非自动运行中
		manulStep:=13;
	ELSE
		errorStep:=5;
		manulStep:=60;
	END_IF
13:
	ctrl_OperCmd.0:=1;
	ctrl_OperCmd.5:=1;// manul 执行
	manulStep:=20;
	
20:
	heatErrorDelayTon(IN:=(NOT status_OperSta.0 OR NOT status_OperSta.5),PT:=errorDelayTime);
	IF heatErrorDelayTon.Q THEN
		//done:=FALSE;
		manuldone:=FALSE;
		errorStep:=6;// 等待AT加热反馈超时
		RETURN;
	END_IF
	heatDoneDelayTon(IN:=status_OperSta.0 OR status_OperSta.5,PT:=doneDelayTimeShortHeat);
	
	IF heatDoneDelayTon.Q THEN
		errorStep:=0;
		manulStep:=30;
		heatErrorDelayTon(IN:=FALSE);
		heatDoneDelayTon(IN:=FALSE);
	END_IF
30:
	IF status_MV=para_Manual_MV THEN//等待AT完成
		errorStep:=0;
		manulStep:=40;
		heatErrorDelayTon(IN:=FALSE);
		heatDoneDelayTon(IN:=FALSE);
	END_IF
	IF status_OutAndAlm.0 OR status_OutAndAlm.1 OR status_OutAndAlm.2 OR status_OutAndAlm.3
	OR status_OutAndAlm.4 OR status_OutAndAlm.5 OR status_OutAndAlm.6 THEN
		errorStep:=3;
		manulStep:=60;
	END_IF
40:
	heatDoneDelayTon(IN:=TRUE,PT:=T#2S);
	IF heatDoneDelayTon.Q THEN
		IF status_MV<=para_Manual_MV THEN
			manulStep:=50;
			heatDoneDelayTon(IN:=FALSE);
		ELSE
			errorStep:=7;//手动控制失控
			manulStep:=60;
		END_IF
	END_IF
50:
	busy:=FALSE;
	manuldone:=TRUE;
60://报错
	ctrl_OperCmd.0:=0;
	ctrl_OperCmd.5:=0;// manul 取消执行
	busy:=FALSE;
	manuldone:=FALSE;
END_CASE
END_ACTION

ACTION Reset_ACT:
IF reset THEN
	IF NOT status_OperSta.0 AND NOT status_OperSta.1 THEN
		busy:=FALSE;
		stop:=FALSE;
		heatting:=FALSE;
	END_IF
	
	//done:=FALSE;
	heatdone:=FALSE;
	ATLdone:=FALSE;
	manuldone:=FALSE;
	errorStep:=0;
	ctrl_OperCmd.0:=0;//停止加热
	ctrl_OperCmd.4:=1;//切换为NOT AT
	ctrl_OperCmd.5:=0;//切换为自动
	heatting:=FALSE;
	reset:=FALSE;
	note_heat:=FALSE;
END_IF

IF stop THEN
	note_heat:=FALSE;
	heatStep:=0;
	atlStep:=0;
	manulStep:=0;
	ctrl_OperCmd.0:=0;//停止加热
	ctrl_OperCmd.4:=1;//切换为NOT AT
	ctrl_OperCmd.5:=0;//切换为自动
	para_SV:=0;//温度设定为0
	IF NOT status_OperSta.0 AND NOT status_OperSta.1 THEN
		busy:=FALSE;
		stop:=FALSE;
		heatting:=FALSE;
	END_IF
END_IF
//100ms保持后复位，模拟上升沿
ATLearRest(IN:=ctrl_OperCmd.2 OR ctrl_OperCmd.4,PT:=T#1S);
IF ATLearRest.Q THEN
	ctrl_OperCmd.2:=0;
	ctrl_OperCmd.4:=0;
END_IF
END_ACTION

ACTION SafeMonitor_ACT:
//notBusyMonitorDelayTon(IN:=NOT busy,PT:=notBusyMonitorDelayTime);
//IF real_TimeMonitor THEN
//	IF notBusyMonitorDelayTon.Q THEN
//		//加热实时检测
//		IF (enableExtAprSw AND NOT extAprSw) AND extRelay THEN
//			errorStep:=1;
//		END_IF

//		IF cylinderType=CylinderType_ButV THEN
//			IF NOT extCondition AND (NOT retdone OR extRelay) THEN//蝶阀单控，检测到开条件消失，强制关闭
//				retract:=TRUE;
//				extRelay:=FALSE;
//			END_IF
//		END_IF
//	END_IF
//END_IF
END_ACTION

ACTION VersionLog:
(*
版本: V1.0.0.0
说明:
	1. 首个版本
	2. 含普通气缸\真空吸类型的控制
	3. 可配置是否有到位信号, 以及到位稳定时间
(--------------------------------------------------)
新版本: V1.0.1.0
更新时间: 2019/11/20 19:00
更新说明:
	1. 优化编写方式
	2. 修改错误编码起始位，现改为从1开始
(--------------------------------------------------)
新版本: V1.0.1.1
更新时间: 2020/03/23 23:00
更新说明:
	1. 优化报错方式
	2. 增加伸出、缩回、复位和停止触发函数
(--------------------------------------------------)
新版本: V1.0.1.2
更新时间: 2020/04/22 09:50
更新说明:
	1. 增加中文报警输出
(--------------------------------------------------)
新版本: V1.0.1.3
更新时间: 2020/09/16
更新说明:
	1. 开放错误ID、错误文本信息获取接口
(--------------------------------------------------)
新版本: V1.0.1.4
更新时间: 2020/10/06
更新说明:
	1. 移除控制模式变量，增加HMI启用条件
	2. 增加外部获取伸出缩回完成信号接口函数
(--------------------------------------------------)
新版本: V1.0.1.5
更新时间: 2020/10/14
更新说明:
	1. 优化代码
(--------------------------------------------------)
*)
END_ACTION

END_FUNCTION_BLOCK

// ---- POUs/BaseModule/ActionModule/OtherModule/ChillerModule.TcPOU
FUNCTION_BLOCK ChillerModule
VAR_INPUT
	condition:BOOL;// 显示条件
	IP:STRING;
	Port: INT;
	alrmmaxTempValue:REAL;// 警告上限
	alrmminTempValue:REAL;// 警告下限
	alrmmaxSpeedValue:REAL;// 警告上限
	alrmminSpeedValue:REAL;// 警告下限
END_VAR
VAR_OUTPUT
	TempValue:REAL;
	SpeedValue:REAL;
	Error:BOOL;
END_VAR
VAR
	changeTempStep	:UDINT;
	readStateStep	:UDINT;
	resetStep		:UDINT;
	startStep		:UDINT;
	stopTempStep	:UDINT;
	
	changeTempBusy	:BOOL;
	readStateBusy	:BOOL;
	resetBusy		:BOOL;
	startBusy		:BOOL;
	stopTempBusy	:BOOL;
	
	changeTempError	:BOOL;
	readStateError	:BOOL;
	resetError		:BOOL;
	startError		:BOOL;
	stopTempError	:BOOL;
	
	
	changeTempDone	:BOOL;
	readStateDone	:BOOL;
	resetDone		:BOOL;
	startDone		:BOOL;
	stopTempDone	:BOOL;
END_VAR

// List
// send
// action

ACTION ACT_ChangeTemp:

END_ACTION

ACTION ACT_ReadState:

END_ACTION

ACTION ACT_Reset:

END_ACTION

ACTION ACT_Start:

END_ACTION

ACTION ACT_Stop:

END_ACTION

END_FUNCTION_BLOCK

// ---- POUs/BaseModule/ActionModule/OtherModule/GaugeViewModule.TcPOU
FUNCTION_BLOCK GaugeViewModule
VAR_INPUT
	inputValue:DINT;// 输入值
	gaugeType:INT;// 类型，1：AIM；2：PSG
	calValueH:REAL;// 计算值上限
	calValueL:REAL;// 计算值下限
	moduleValueH:REAL;// 模块上限
	moduleValueL:REAL;// 模块下限
	alrmmaxValue:REAL;// 警告上限
	alrmminValue:REAL;// 警告下限
	condition:BOOL;// 显示条件
	initString:STRING:='-----';// 初始显示字符串：*****
END_VAR
VAR_OUTPUT
	outputValue:REAL;
	outputValue_String:STRING;
	error:BOOL;
END_VAR
VAR
	factor:REAL;// 转换因子
	temp:REAL;
	test:REAL;
	tT:TON;
END_VAR

IF ((moduleValueH-moduleValueL)>0.0) THEN
	factor:=(calValueH-calValueL)/(moduleValueH-moduleValueL);
	temp:=factor*DINT_TO_REAL(inputValue);
	IF gaugeType=1 THEN
		test:=(7.0*temp/8.0-10.75);
		outputValue:=LREAL_TO_REAL(EXPT(10,test));
//		outputValue_String:=REAL_TO_STRING(outputValue);
		Real_e(inputReal:=outputValue,outputString=>outputValue_String);
	ELSE
		test:=(temp-2.448)/1.286;
		outputValue:=LREAL_TO_REAL(EXPT(10,test));
		outputValue_String:=Real_2f(realStr:=REAL_TO_STRING(outputValue));
	END_IF
	tT(IN:=NOT (( outputValue>alrmminValue) AND inputValue>10),PT:=T#2S);
	IF tT.Q THEN
		error:=TRUE;
	ELSE
		error:=FALSE;
	END_IF
	
	IF condition THEN
		;
	ELSE
		outputValue_String:=initString;
	END_IF
END_IF

METHOD Real_2f : STRING
VAR_INPUT
	realStr:STRING;
END_VAR
VAR
	decimalPlaces:INT:=1;
	dotPos : INT;
END_VAR
dotPos := FIND(realStr, '.');

IF dotPos > 0 THEN
    // 截取小数点后指定位数
    realStr := LEFT(realStr, dotPos + decimalPlaces);
END_IF
Real_2f:=realStr;
END_METHOD

METHOD Real_e : BOOL
VAR_INPUT
	inputReal : REAL; // 输入：REAL 类型数据
END_VAR
VAR_OUTPUT
	outputString : STRING(50);    // 输出：科学计数法表示的 STRING 数据
END_VAR
VAR
	tempString : STRING(50);       // 临时字符串变量
    mantissaPart : STRING(20);     // 尾数部分
    exponentValue : INT;           // 指数值
    decimalPointPos : INT;         // 小数点位置
	posP:INT;// 整数部分
    isNegative : BOOL := FALSE;    // 是否为负数
	i:INT;
	endFlag:BOOL;
	maxPos:INT:=20;
	tempReal:REAL;
	tempReal1:REAL;
	temstr:STRING;
	decimalPlaces:INT:=1;
	dotPos : INT;
END_VAR
 // Step 1: 处理负数
 endFlag:=FALSE;
IF inputReal>1.0 THEN
	outputString:=REAL_TO_STRING(inputReal);
	RETURN;
END_IF
IF inputReal < 0 THEN
    isNegative := TRUE;
    inputReal := ABS(inputReal); // 取绝对值
END_IF

tempReal:=inputReal;
FOR i:=1 TO maxPos DO
	tempReal:=tempReal*10.0;
	posP:=REAL_TO_INT(tempReal)/10;
	tempReal1:=REAL_TO_INT(tempReal*10.0)/100.0;
	IF posP<>0 THEN
		exponentValue:=i;
		endFlag:=TRUE;
		i:=20;
	END_IF
END_FOR

//// Step 5: 提取尾数部分
//IF decimalPointPos > 0 THEN
//	mantissaPart :=CONCAT(mantissaPart,LEFT(tempString, 1));
//	mantissaPart :=CONCAT(mantissaPart,'.');
//	mantissaPart :=CONCAT(mantissaPart,MID(tempString, 2, LEN(tempString) - 1));
//ELSE
//    mantissaPart := tempString; // 如果没有小数点，直接使用原字符串
//END_IF

// Step 6: 构建底数为 10 的表达式
temstr:=REAL_TO_STRING(tempReal1);
dotPos := FIND(temstr, '.');

IF dotPos > 0 THEN
    // 截取小数点后指定位数
    temstr := LEFT(temstr, dotPos + decimalPlaces);
END_IF

IF isNegative THEN
	outputString :=CONCAT(outputString,'-');
	outputString :=CONCAT(outputString,temstr);
	outputString :=CONCAT(outputString,' * 10^');
	outputString :=CONCAT(outputString,INT_TO_STRING(exponentValue));
ELSE
	outputString :=CONCAT(outputString,temstr);
	outputString :=CONCAT(outputString,' * 10^-');
	outputString :=CONCAT(outputString,INT_TO_STRING(exponentValue-1));
END_IF

// 输出结果
// outputString 现在包含底数为 10 的表达式
END_METHOD

END_FUNCTION_BLOCK

// ---- POUs/BaseModule/ActionModule/OtherModule/ChamberGaugeViewModule.TcPOU
FUNCTION_BLOCK ChamberGaugeViewModule
VAR_INPUT
	inputValue:DINT;// 输入值
	gaugeType:INT;// 类型，1：AIM；2：PSG
	calValueH:REAL;// 计算值上限
	calValueL:REAL;// 计算值下限
	moduleValueH:REAL;// 模块上限
	moduleValueL:REAL;// 模块下限
	alrmmaxValue:REAL;// 警告上限
	alrmminValue:REAL;// 警告下限
	condition:BOOL;// 显示条件
	initString:STRING:='-----';// 初始显示字符串：*****
END_VAR
VAR_OUTPUT
	outputValue:REAL;
	outputValue1:REAL;
	outputValue_String:STRING;
	error:BOOL;
END_VAR
VAR
	factor:REAL;// 转换因子
	temp:REAL;
	test:REAL;
	tT:TON;
END_VAR

IF ((moduleValueH-moduleValueL)>0.0) THEN
	factor:=(calValueH-calValueL)/(moduleValueH-moduleValueL);
	temp:=factor*DINT_TO_REAL(inputValue);
	outputValue:=temp*((alrmmaxValue-alrmminValue)/(19-4));
//	IF outputValue<100000 THEN
//		outputValue_String:=REAL_TO_STRING(outputValue-1100);
//		outputValue1:=(outputValue-1100);
//	ELSE
//		outputValue_String:=REAL_TO_STRING(outputValue);
//		outputValue1:=(outputValue);
//	END_IF
	IF outputValue-1100<1 THEN
		outputValue:=1112.4;
	END_IF
	outputValue_String:=REAL_TO_STRING(outputValue-1100);
	outputValue1:=(outputValue-1100);
	tT(IN:=NOT (( outputValue>alrmminValue) AND inputValue>10),PT:=T#2S);
	IF tT.Q THEN
		error:=TRUE;
	ELSE
		error:=FALSE;
	END_IF
	
	IF condition THEN
		;
	ELSE
		outputValue_String:=initString;
	END_IF
END_IF

END_FUNCTION_BLOCK

// ---- POUs/BaseModule/COE/EcCoeSdo_ForTest.TcPOU
PROGRAM EcCoeSdo_ForTest
VAR_INPUT
	bWrite:BOOL;
	bRead:BOOL;
	nEncoderResolution_Write:DINT:=525;//编码器分辨率
	bWrite2:BOOL;
	bRead2:BOOL;
	nEncoderResolution_Write2:DINT:=1100;//编码器分辨率
END_VAR
VAR_OUTPUT
	nEncoderResolution_Read:DINT;//编码器分辨率
	nEncoderResolution_Read2:DINT;//编码器分辨率
END_VAR
VAR
	fbECCOE_READ_WRITE:FB_ECCOE_READ_WRITE;
	fbECCOE_READ_WRITE2:FB_ECCOE_READ_WRITE;
	tInit:TON;
	t1:TON;
END_VAR

tInit(IN:= TRUE, PT:= T#10S, Q=> , ET=> );
IF NOT tInit.Q THEN
	RETURN;
END_IF

IF bWrite THEN
	bWrite:=FALSE;
	fbECCOE_READ_WRITE.Act_Write();
END_IF
IF bRead THEN
	bRead:=FALSE;
	fbECCOE_READ_WRITE.Act_Read();
END_IF
fbECCOE_READ_WRITE(
	sNetId:= '5.57.12.34.3.1', 
	nSlaveAddr:= 1009, 
	nIndex:= 16#20E4, 
	nSubIndex:= 0, 
	pReadBuff:= ADR(nEncoderResolution_Read), 
	cbReadBuffLen:= SIZEOF(nEncoderResolution_Read), 
	pWriteBuff:= ADR(nEncoderResolution_Write), 
	cbWriteBuffLen:= SIZEOF(nEncoderResolution_Write), 
	bBusy=> , 
	bDone=> , 
	bError=> , 
	nErrId=> );
	
//
IF bWrite2 THEN
	bWrite2:=FALSE;
	fbECCOE_READ_WRITE2.Act_Write();
END_IF
IF bRead2 THEN
	bRead2:=FALSE;
	fbECCOE_READ_WRITE2.Act_Read();
END_IF
fbECCOE_READ_WRITE2(
	sNetId:= '5.57.12.34.3.1', 
	nSlaveAddr:= 1010, 
	nIndex:= 16#20E4, 
	nSubIndex:= 0, 
	pReadBuff:= ADR(nEncoderResolution_Read2), 
	cbReadBuffLen:= SIZEOF(nEncoderResolution_Read2), 
	pWriteBuff:= ADR(nEncoderResolution_Write2), 
	cbWriteBuffLen:= SIZEOF(nEncoderResolution_Write2), 
	bBusy=> , 
	bDone=> , 
	bError=> , 
	nErrId=> );
	
t1(IN:= NOT t1.Q AND NOT fbECCOE_READ_WRITE.bBusy, PT:= T#500MS, Q=> , ET=> );
IF t1.Q THEN
	fbECCOE_READ_WRITE.Act_Read();
	fbECCOE_READ_WRITE2.Act_Read();
END_IF

END_PROGRAM

// ---- POUs/BaseModule/COE/FB_ECCOE_READ_WRITE.TcPOU
FUNCTION_BLOCK FB_ECCOE_READ_WRITE
VAR_INPUT
	sNetId      			: T_AmsNetId:= '';//I/O->Devices->Device 1(EtherCAT)-->EtherCAT选项卡->NetId
    nSlaveAddr  			: UINT;//I/O->Devices->Device 1(EtherCAT)-->选中对应的驱动器(例如Drive 20)->EtherCAT选项卡->EtherCAT Addr
    nIndex					: WORD := 0;//待读写的参数索引
	nSubIndex      			: BYTE;//待读写的参数索引的子索引
    pReadBuff     			: PVOID;//待读的数据缓存
	cbReadBuffLen			: UDINT;//待读的数据缓存长度；使用sizeof
    pWriteBuff     			: PVOID;//待写的数据缓存
	cbWriteBuffLen			: UDINT;//待写的数据缓存长度：使用sizeof
END_VAR
VAR_OUTPUT
	bBusy					: BOOL;
	bDone					: BOOL;
    bError      			: BOOL;
    nErrId      			: UDINT;
END_VAR
VAR
	fbEcCoeSdoRead  		: FB_EcCoeSdoRead;
	fbEcCoeSdoWrite  		: FB_EcCoeSdoWrite;
	ftrig_Busy				: F_TRIG;
	f2trig_Busy				: F_TRIG;
	f3trig_Busy				: F_TRIG;
END_VAR

fbEcCoeSdoRead(
	sNetId:= sNetId, 
	nSlaveAddr:= nSlaveAddr, 
	nSubIndex:= nSubIndex, 
	nIndex:= nIndex, 
	pDstBuf:= pReadBuff, 
	cbBufLen:= cbReadBuffLen, 
	bExecute:= , 
	tTimeout:= , 
	bBusy=> , 
	bError=> , 
	nErrId=> );
fbEcCoeSdoWrite(
	sNetId:= sNetId, 
	nSlaveAddr:= nSlaveAddr, 
	nSubIndex:= nSubIndex, 
	nIndex:= nIndex, 
	pSrcBuf:= pWriteBuff, 
	cbBufLen:= cbWriteBuffLen, 
	bExecute:= , 
	tTimeout:= , 
	bBusy=> , 
	bError=> , 
	nErrId=> );

bBusy:=fbEcCoeSdoRead.bBusy OR fbEcCoeSdoWrite.bBusy;
bError:=fbEcCoeSdoRead.bError OR fbEcCoeSdoWrite.bError;
IF fbEcCoeSdoRead.bError THEN
	nErrId:=fbEcCoeSdoRead.nErrId;
ELSIF fbEcCoeSdoWrite.bError THEN
	nErrId:=fbEcCoeSdoWrite.nErrId;
ELSE
	nErrId:=0;
END_IF
ftrig_Busy(CLK:= bBusy, Q=> );
IF bBusy THEN
	bDone:=FALSE;
END_IF
IF NOT bError AND ftrig_Busy.Q THEN
	bDone:=TRUE;
END_IF
f2trig_Busy(CLK:= fbEcCoeSdoRead.bBusy, Q=> );
IF f2trig_Busy.Q THEN
	fbEcCoeSdoRead(bExecute:=FALSE);
END_IF
f3trig_Busy(CLK:= fbEcCoeSdoWrite.bBusy, Q=> );
IF f3trig_Busy.Q THEN
	fbEcCoeSdoWrite(bExecute:=FALSE);
END_IF

METHOD Act_Read : BOOL
VAR_INPUT
END_VAR
fbEcCoeSdoRead(bExecute:=FALSE);

fbEcCoeSdoRead(bExecute:=TRUE);

bDone:=FALSE;
Act_Read:=TRUE;
END_METHOD

METHOD Act_Write : BOOL
VAR_INPUT
END_VAR
fbEcCoeSdoWrite(bExecute:=FALSE);

fbEcCoeSdoWrite(bExecute:=TRUE);

bDone:=FALSE;
Act_Write:=TRUE;
END_METHOD

END_FUNCTION_BLOCK

// ---- POUs/BaseModule/Communication/FuncModule_RS232_Byte.TcPOU
PROGRAM FuncModule_RS232_Byte
VAR_INPUT
	serialExcute				:BOOL;// RS485开始一次参数读取
	serialSlaveID				:UINT;// 485从站节点号
END_VAR
VAR_OUTPUT
	serialBusy						:BOOL;
	serialDone						:BOOL;
	serialError						:BOOL;
	temperature				:REAL;//分子泵温度
	current					:REAL;//分子泵电流
	speed					:REAL;//分子泵转速
END_VAR
VAR
	currentTemp:INT;// 电流中转变量
	temperatureTemp				:DINT;// 温度中转变量
	speedTemp					:DINT;// 速度中转变量
	(*
	 *xBuffer 的作用是，在 PLC 要发送的数据和串行通讯的硬件 Process Data 之间设置一个缓存区。
	 *比如 KL6outData22B 类型的接口，每个 PLC 周期只能发送 22 字节。假如程序需要发送的数据为 100 个，
	 *那么实际上 PLC 程序是把这些数据放到 TxBuffer 中，再由硬件分几个 PLC 周期发送出去
	*)
	TxBuffer_TMP:					ComBuffer;		
	RxBuffer_TMP:					ComBuffer;
	
	COMin				AT%I*		:KL6inData22B;		
	COMout				AT%Q*		:KL6outData22B;
		
	COMportControl					:SerialLineControl;
	
	//Byte方式
	send1:							SendData;
	receive1:						ReceiveData;
 
	Timer1:							TON;
	t1:								TON;
	ITemp:INT;
	
	nSendByteLength: 				UDINT:= 11;	//发送数据的长度
	arr_SendData:					ARRAY[1..20]			OF		BYTE;(*READ*)//发送数据
	arr_RcvData:					ARRAY[1..200]			OF		BYTE;//接受数据
	arr_RcvData_Temp:				ARRAY[1..200]			OF		BYTE;//接受数据中转
	arr_RcvData_Clear:				ARRAY[1..200]			OF		BYTE;//接受数据清空
	arr_Temp:						ARRAY [1..2] OF BYTE;//高低位互换
	arr_Temp1:						ARRAY [1..2] OF BYTE;//高低位互换
	serialStep						:UINT;				//处理步数
	serialErrorID					:UINT;
	serialTimeOut:BOOL;//接收数据超时
	serialRecError:BOOL;//接收数据错误
	testReal:REAL;
	strTemp:STRING;
	//字符串方式
	(*send1:							SendString;
	receive1:						ReceiveString;
	
	Timer1:							TON;
	
	_sendString:					STRING:='4567';
	_receive1string:				STRING;
	_recvLast:						STRING;				//保存上一个周期接收的字符*)
	
END_VAR

(*
 *功能块的作用，把 TxBuffer 缓存区的数据经过 Process Data 的 ComOut 发送出去，
 *而把 ComIn 中的数据接收到 RxBuffer。引用这个功能块的程序执行周期越短，
 *数据交换的效率就越高，所以这段程序应该放在快速任务中作为 Backgroud 代码无条件执行。
*)
COMportControl(
	Mode:= SERIALLINEMODE_KL6_22B_STANDARD, 
	pComIn:= ADR(COMin), 
	pComOut:= ADR(COMout), 
	SizeComIn:= SIZEOF(COMin), 
	Error=> , 
	ErrorID=> , 
	TxBuffer:= TxBuffer_TMP, 
	RxBuffer:= RxBuffer_TMP );
IF receive1.Error <> COMERROR_NOERROR THEN
	serialRecError:=TRUE;
END_IF
receive1(
	pPrefix:= , 
	LenPrefix:= , 
	pSuffix:= , 
	LenSuffix:= , 
	pReceiveData:= ADR(arr_RcvData), 
	SizeReceiveData:= 100, 
	Timeout:= T#100MS, //临时设置成10S调试用
	Reset:= , 
	DataReceived=> , 
	busy=> , 
	Error=> , 
	RxTimeout=> , 
	LenReceiveData=> , 
	RXbuffer:= RxBuffer_TMP);
//testReal:=BYTE_TO_REAL(arr_RcvData_Temp);
CASE serialStep OF
	0:
	IF serialExcute THEN
		serialExcute:=FALSE;
		IF NOT serialBusy THEN
			serialStep:=10;
			serialBusy:=TRUE;
			serialDone:=FALSE;
			serialError:=FALSE;
			serialTimeOut:=FALSE;
			serialRecError:=FALSE;
			receive1(//复位
				pPrefix:= , 
				LenPrefix:= , 
				pSuffix:= , 
				LenSuffix:= , 
				pReceiveData:= , 
				SizeReceiveData:=, 
				Timeout:= T#300MS, 
				Reset:= , 
				DataReceived=> , 
				busy=> , 
				Error=> , 
				RxTimeout=> , 
				LenReceiveData=> , 
				RXbuffer:= RxBuffer_TMP);
		END_IF
	END_IF
	Timer1(IN:= FALSE);
	;
	10:
		//第二和第三位代表ID号
		arr_SendData[1]	:=16#40;
		IF serialSlaveID<16 THEN
			arr_SendData[2]:=F_ToASC(str:='0');
			arr_SendData[3]:=F_ToASC(str:=CalASII_Str(serialSlaveID));
		ELSE
			arr_SendData[2]:=F_ToASC(str:=CalASII_Str(serialSlaveID/16));
			arr_SendData[3]:=F_ToASC(str:=CalASII_Str(serialSlaveID MOD 16));
		END_IF
		arr_SendData[4]:=16#02;
		arr_SendData[5]:=16#30;
		arr_SendData[6]:=16#30;
		arr_SendData[7]:=16#31;
		arr_SendData[8]:=16#3F;
		arr_SendData[9]:=16#5B;
		arr_SendData[10]:=16#03;
		arr_SendData[11]:=16#AB;
		serialStep:=100;
	100:
		send1(
			pSendData:= ADR(arr_SendData), 
			Length:= nSendByteLength, 
			Busy=> , 
			Error=> , 
			TXbuffer:= TxBuffer_TMP);
		serialStep:=serialStep+20;
	110:
		Timer1(IN:= NOT timer1.q, PT:=T#00MS);
		IF Timer1.Q THEN
			serialStep:=serialStep+10;
			Timer1(IN:= FALSE);
		END_IF
	120:
		Timer1(IN:= NOT timer1.q, PT:=T#50000MS);
		IF Timer1.Q THEN
			serialStep:=6000;
			Timer1(IN:= FALSE);
			serialTimeOut:=TRUE;
			RETURN;
		END_IF
		IF NOT receive1.busy  THEN
			Timer1(IN:= FALSE);
			serialTimeOut:=FALSE;
			serialStep:=200;
		END_IF
		IF receive1.Error <> COMERROR_NOERROR THEN
			serialRecError:=TRUE;
		END_IF
	200://数据处理
		arr_RcvData_Temp:=arr_RcvData;
		arr_RcvData:=arr_RcvData_Clear;
		serialStep:=serialStep+10;
	210:
		//第二和第三位代表ID号;看情况决定是否需要判断节点反馈的节点号
		IF NOT receive1.DataReceived THEN
			serialStep:=serialStep+10;
			Timer1(IN:= FALSE);
		END_IF
	220:
		//数据转换
		Timer1(IN:= FALSE);
		serialStep:=1000;
	
	1000:
		Timer1(IN:= NOT timer1.q, PT:=T#1000MS);
		IF Timer1.Q THEN
			serialStep:=10;
			Timer1(IN:= FALSE);
			serialTimeOut:=TRUE;
		END_IF
	;
	5000://done
		serialBusy:=FALSE;
		serialDone:=TRUE;
		serialError:=FALSE;
		serialStep:=0;
	;
	6000://error
		serialBusy:=FALSE;
		serialDone:=FALSE;
		serialError:=TRUE;
		serialStep:=0;
	;
	
END_CASE

METHOD CalASII_Str : STRING
VAR_INPUT
	date1:UINT;
END_VAR
IF date1=10 THEN
	CalASII_Str:='A';
END_IF
IF date1=11 THEN
	CalASII_Str:='B';
END_IF
IF date1=12 THEN
	CalASII_Str:='C';
END_IF
IF date1=13 THEN
	CalASII_Str:='D';
END_IF
IF date1=14 THEN
	CalASII_Str:='E';
END_IF
IF date1=15 THEN
	CalASII_Str:='F';
END_IF
IF date1<10 THEN
	CalASII_Str:=UINT_TO_STRING(date1);
END_IF
IF date1>15 THEN
	CalASII_Str:=UINT_TO_STRING(date1);
END_IF
END_METHOD

END_PROGRAM

// ---- POUs/BaseModule/Communication/FuncModule_TCPIP_Binary_POU.TcPOU
PROGRAM FuncModule_TCPIP_Binary_POU
VAR_INPUT
	nSocketType:UINT:=0;// socket 类型; 0 表示 server; 1 表示 client;
	sTerminalName:STRING;// 通讯对方名称 自定义
	sHost:STRING(20):='127.0.0.1';// 通讯IP地址; server时表示本地host; client时表示远程host
	nPort:UDINT:=8900;// 通讯端口号;
	bEnable:BOOL:=TRUE;// 通讯启用\禁用连接
	nQueueInterval:UDINT:=50;// 发送队列时间间隔 单位ms
	logHandleArray:ARRAY [1..5] OF POINTER TO printLogModule_EX;// log 操作 handle 数组
	logHandleArrayLength:UINT:=0;// log 操作 handle 数组长度, 不超过5
	enHeartBeat:BOOL;// 启用心跳包命令
	cmdHeartBeat:DINT;// 心跳包命令
END_VAR
VAR_OUTPUT
	bSendCondition	:BOOL;//可发送条件
	bSocketConnected:BOOL;//连接状态
END_VAR
VAR CONSTANT
	cNumBegin		:DINT:=1;
	cNumEnd			:DINT:=100;
END_VAR
VAR
	sendDataArray	:ARRAY [cNumBegin..cNumEnd] OF struct_Tester;
	length			:DINT:=0;
	endPoint		:DINT:=cNumBegin;
	popupSendData	:struct_Tester;
	//popup
	popupStep		:UINT:=0;
	popupTON1		:TON;
	popupTON2		:TON;
	iPopup			:DINT:=0;
	_PopupLength	:DINT:=0;
END_VAR
VAR
	tcpipClient					:tcpipClientModule_EX;
	tcpipServer					:tcpipServerModule_EX;////定义服务器对象
	
	tcpipSendDataBuff_Server	:ST_TCPIP_DATA_STRUCT_ALC;//发送数据 Buff server
	tcpipSendDataBuff_Client	:ST_TCPIP_DATA_STRUCT_ALC;//发送数据 Buff client
	
	tcpipSendDataClear			:ST_TCPIP_DATA_STRUCT_ALC;//发送数据 清空
	tcpipSendData				:ST_TCPIP_DATA_STRUCT_ALC;//发送数据
	
	tcpipRecDataBuff_Server		:ST_TCPIP_DATA_STRUCT_ALC;//已接收数据 Buff server
	tcpipRecDataBuff_Client		:ST_TCPIP_DATA_STRUCT_ALC;//已接收数据 Buff client
	
	tcpipRecDataClear			:ST_TCPIP_DATA_STRUCT_ALC;//已接收数据 清空
	tcpipRecData				:ST_TCPIP_DATA_STRUCT_ALC;//已接收数据
	
	tcpConnectR_Trig			:R_Trig;//初始连接上升沿
	tcpConnectF_Trig			:F_Trig;//初始连接下降沿
	registerStep				:UDINT;//ALC注册控制步
	registerTON					:TON;//ALC注册延时
	
	logHandleArray_index		:UINT:=1;
END_VAR


CASE nSocketType OF
0://TCPIP server
	tcpipServer(
		sSrvNetId:= , 
		sLocalHost:=sHost , 
		nLocalPort:=nPort , 
		bStartConnect:=bEnable , 
		tcpipSDataLen:=SIZEOF(tcpipSendDataBuff_Server) , 
		tcpipSData:=ADR(tcpipSendDataBuff_Server) , 
		bSend:= , 
		tcpipRecDataLen:=SIZEOF(tcpipRecDataBuff_Server) , 
		tcpipRecData:=ADR(tcpipRecDataBuff_Server) , 
		bAccepted=> , 
		bSendBusy=> , 
		bRecData=> );
	bSendCondition:=tcpipServer.bAccepted AND NOT tcpipServer.bSendBusy;
	//TCPIP连接
	bSocketConnected:=tcpipServer.bAccepted;
	IF NOT tcpipServer.bAccepted THEN
		length:=0;
		endPoint:=cNumBegin;
	END_IF
	tcpConnectR_Trig(CLK:=tcpipServer.bAccepted);
	tcpConnectF_Trig(CLK:=tcpipServer.bAccepted);

1://TCPIP client
	tcpipClient(
		sSrvNetId:= , 
		sRemoteHost:=sHost , 
		nRemotePort:=nPort , 
		bStartConnect:=bEnable , 
		tcpipSDataLen:=SIZEOF(tcpipSendDataBuff_Client) , 
		tcpipSData:=ADR(tcpipSendDataBuff_Client) , 
		bSend:= , 
		tcpipRecDataLen:=SIZEOF(tcpipRecDataBuff_Client) , 
		tcpipRecData:=ADR(tcpipRecDataBuff_Client) , 
		bConnected=> , 
		bSendBusy=> , 
		bRecData=> );
	bSendCondition:=tcpipClient.bConnected AND NOT tcpipClient.bSendBusy;
	//TCPIP连接
	bSocketConnected:=tcpipClient.bConnected;
	IF NOT tcpipClient.bConnected THEN
		length:=0;
		endPoint:=cNumBegin;
	END_IF
	tcpConnectR_Trig(CLK:=tcpipClient.bConnected);
	tcpConnectF_Trig(CLK:=tcpipClient.bConnected);
END_CASE

IF tcpConnectR_Trig.Q THEN
	FOR logHandleArray_index:=1 TO logHandleArrayLength DO
		logHandleArray[logHandleArray_index]^.append(CONCAT(sTerminalName, ' has been connected'));
	END_FOR
	registerStep:=10;
END_IF
IF tcpConnectF_Trig.Q THEN
	FOR logHandleArray_index:=1 TO logHandleArrayLength DO
		logHandleArray[logHandleArray_index]^.append(CONCAT(sTerminalName, ' has been disconnected'));
	END_FOR
	registerStep:=0;
END_IF
//数据接收处理
CASE nSocketType OF
0://TCPIP server
	IF tcpipServer.bRecData THEN
		tcpipRecData:=tcpipRecDataBuff_Server;//buff转存
		tcpipRecDataBuff_Server:=tcpipRecDataClear;//转存之后清空buff
		dataProcessing();
	END_IF
1://TCPIP client
	IF tcpipClient.bRecData THEN
		tcpipRecData:=tcpipRecDataBuff_Client;//buff转存
		tcpipRecDataBuff_Client:=tcpipRecDataClear;//转存之后清空buff
		dataProcessing();
	END_IF
END_CASE


popup();

CASE registerStep OF
0:
	//Ready
END_CASE

METHOD appendSend : BOOL
VAR_INPUT
	channel		:DINT;
	msgType		:DINT:=0;
	funCode		:DINT;
	value1		:REAL:=0;
	value2		:REAL:=0;
	value3		:REAL:=0;
	value4		:REAL:=0;
	value5		:REAL:=0;
	errID		:LINT:=0;
	str			:STRING(g_nMaxByte_Client):='';
END_VAR

IF endPoint>(cNumEnd-1) THEN
	RETURN;
END_IF
sendDataArray[endPoint].channel:=channel;
sendDataArray[endPoint].msgType:=msgType;
sendDataArray[endPoint].funCode:=funCode;
sendDataArray[endPoint].msgType:=msgType;
sendDataArray[endPoint].value1:=value1;
sendDataArray[endPoint].value2:=value2;
sendDataArray[endPoint].value3:=value3;
sendDataArray[endPoint].value4:=value4;
sendDataArray[endPoint].value5:=value5;
sendDataArray[endPoint].errID:=errID;
sendDataArray[endPoint].str:=str;

endPoint:=endPoint+1;
length:=endPoint-cNumBegin;
END_METHOD

METHOD dataProcessing : BOOL
VAR_INPUT
END_VAR
FOR logHandleArray_index:=1 TO logHandleArrayLength DO
	CASE nSocketType OF
	0://TCPIP server
		IF enHeartBeat AND tcpipRecData.funCode=cmdHeartBeat THEN// 不打印心跳包命令
			EXIT;
		END_IF
		logHandleArray[logHandleArray_index]^.append(CONCAT(CONCAT(CONCAT('Recevie From ', sTerminalName), ' -- '),ALCData2String(tcpipRecData)));
	1://TCPIP client
		IF enHeartBeat AND tcpipRecData.funCode=cmdHeartBeat THEN// 不打印心跳包命令
			EXIT;
		END_IF
		logHandleArray[logHandleArray_index]^.append(CONCAT(CONCAT(CONCAT('Recevie From ', sTerminalName), ' -- '),ALCData2String(tcpipRecData)));
	END_CASE
END_FOR

appendSend(1,1,23,0,9.9,0,0,0,88,'1213adf');
CASE tcpipRecData.msgType OF
0://对方请求
	CASE tcpipRecData.funCode OF
	(*RotateStart_TM:
		gRotateStart_TM_Trig:=TRUE;
		gRotateStart_TM_SetVelo:=TO_LREAL(tcpipRecData.value1);
		Rotate_Start_POU.func_reset_status();
		Rotate_Start_POU.trigger:=TRUE;
		
		IF 0=tcpipRecData.errID THEN
			;
		ELSE
			;
		END_IF
		//appendSend(0,1,tcpipRecData.funCode,0.0,0.0,0.0,0.0,0.0,0,'');
	
	RotateStop_TM:
		IF 0=tcpipRecData.errID THEN
			;
		ELSE
			;
		END_IF
		//appendSend(0,1,tcpipRecData.funCode,0.0,0.0,0.0,0.0,0.0,0,'');
	*)
	END_CASE
1://对方响应
	CASE tcpipRecData.funCode OF
	(*LoadDUT_TM:
		IF 0=tcpipRecData.errID THEN
			;
		ELSE
			;
		END_IF
	Error_TM:
		IF 0=tcpipRecData.errID THEN
			;
		ELSE
			;
		END_IF
	*)
	END_CASE
END_CASE
END_METHOD

METHOD PRIVATE popup : BOOL
VAR_INPUT
END_VAR
CASE popupStep OF
0:
	IF length>0 AND bSendCondition THEN
		_PopupLength:=length;
		popupSendData:=sendDataArray[cNumBegin];
		FOR iPopup:=cNumBegin TO (_PopupLength-1) DO
			sendDataArray[iPopup]:=sendDataArray[iPopup+1];
		END_FOR
		endPoint:=endPoint-1;
		length:=endPoint-cNumBegin;
		sendData(popupSendData);//此处是调用信息发送
		popupStep:=10;
	END_IF
10:
	popupTON2(IN:=NOT popupTON2.Q, PT:=T#2S);
	IF NOT bSendCondition OR popupTON2.Q THEN
		popupTON2(IN:=FALSE);
		popupStep:=11;
	END_IF
11:
	IF bSendCondition THEN
		popupStep:=12;
	END_IF
	popupTON1(IN:=FALSE);
12:
	//popupTON1(IN:=NOT popupTON1.Q,PT:=T#10MS);
	popupTON1(IN:=NOT popupTON1.Q,PT:=TO_TIME(nQueueInterval));
	IF popupTON1.Q THEN
		popupStep:=0;
	END_IF
END_CASE
END_METHOD

METHOD PRIVATE sendData : BOOL
VAR_INPUT
	dataStruct	:struct_Tester;
END_VAR
IF bSendCondition AND bEnable THEN
	tcpipSendData.channel	:=dataStruct.channel;
	tcpipSendData.msgType	:=dataStruct.msgType;
	tcpipSendData.funCode	:=dataStruct.funCode;
	tcpipSendData.value1	:=dataStruct.value1;
	tcpipSendData.value2	:=dataStruct.value2;
	tcpipSendData.value3	:=dataStruct.value3;
	tcpipSendData.value4	:=dataStruct.value4;
	tcpipSendData.value5	:=dataStruct.value5;
	tcpipSendData.errID		:=dataStruct.errID;
	tcpipSendData.str		:=tcpipServer.string2ASCII(dataStruct.str);
	
	CASE nSocketType OF
	0://TCPIP server
		tcpipSendDataBuff_Server:=tcpipSendData;
		tcpipSendData:=tcpipSendDataClear;	
		tcpipServer.bSend:=TRUE;
	1://TCPIP client
		tcpipSendDataBuff_Client:=tcpipSendData;
		tcpipSendData:=tcpipSendDataClear;	
		tcpipClient.bSend:=TRUE;
	END_CASE
	
	FOR logHandleArray_index:=1 TO logHandleArrayLength DO
		CASE nSocketType OF
		0://TCPIP server
			IF enHeartBeat AND dataStruct.funCode=cmdHeartBeat THEN// 不打印心跳包命令
				EXIT;
			END_IF
			logHandleArray[logHandleArray_index]^.append(CONCAT(CONCAT(CONCAT('Send To ', sTerminalName), ' -- '),ALCData2String(tcpipSendDataBuff_Server)));
		1://TCPIP client
			IF enHeartBeat AND dataStruct.funCode=cmdHeartBeat THEN// 不打印心跳包命令
				EXIT;
			END_IF
			logHandleArray[logHandleArray_index]^.append(CONCAT(CONCAT(CONCAT('Send To ', sTerminalName), ' -- '),ALCData2String(tcpipSendDataBuff_Client)));
		END_CASE
	END_FOR
END_IF
END_METHOD

END_PROGRAM

// ---- POUs/BaseModule/Communication/FuncModule_TCPIP_String_POU.TcPOU
PROGRAM FuncModule_TCPIP_String_POU
VAR_INPUT
	nSocketType:UINT:=0;// socket 类型; 0 表示 server; 1 表示 client;
	sTerminalName:STRING;// 通讯对方名称 自定义
	sHost:STRING(20):='127.0.0.1';// 通讯IP地址; server时表示本地host; client时表示远程host
	nPort:UDINT:=8900;// 通讯端口号;
	bEnable:BOOL:=TRUE;// 通讯启用\禁用连接
	sSendSuffix:STRING:='';//此处可统一添加发送后缀字符 $R$N
	nQueueInterval:UDINT:=50;// 发送队列时间间隔 单位ms
	logHandleArray:ARRAY [1..5] OF POINTER TO printLogModule_EX;// log 操作 handle 数组
	logHandleArrayLength:UINT:=0;// log 操作 handle 数组长度, 不超过5
END_VAR
VAR_OUTPUT
	bSendCondition	:BOOL;//可发送条件
	bSocketConnected:BOOL;//连接状态
END_VAR
VAR CONSTANT
	cNumBegin		:DINT:=1;
	cNumEnd			:DINT:=100;
END_VAR
VAR
	sendDataArray	:ARRAY [cNumBegin..cNumEnd] OF STRING(255);
	length			:DINT:=0;
	endPoint		:DINT:=cNumBegin;
	popupSendData	:STRING(255);
	//popup
	popupStep		:UINT:=0;
	popupTON1		:TON;
	popupTON2		:TON;
	iPopup			:DINT:=0;
	_PopupLength	:DINT:=0;
END_VAR
VAR
	tcpipClient					:tcpipClientModule_EX;
	tcpipServer					:tcpipServerModule_EX;////定义服务器对象
	
	tcpipSendDataBuff_Server	:STRING(255);//发送数据 Buff server
	tcpipSendDataBuff_Client	:STRING(255);//发送数据 Buff client
	
	tcpipSendDataClear			:STRING(255);//发送数据 清空
	tcpipSendData				:STRING(255);//发送数据
	
	tcpipRecDataBuff_Server		:STRING(255);//已接收数据 Buff server
	tcpipRecDataBuff_Client		:STRING(255);//已接收数据 Buff client
	
	tcpipRecDataClear			:STRING(255);//已接收数据 清空
	tcpipRecData				:STRING(255);//已接收数据
	
	tcpConnectR_Trig			:R_Trig;//初始连接上升沿
	tcpConnectF_Trig			:F_Trig;//初始连接下降沿
	registerStep				:UDINT;//ALC注册控制步
	registerTON					:TON;//ALC注册延时
	
	logHandleArray_index		:UINT:=1;
END_VAR


CASE nSocketType OF
0://TCPIP server
	tcpipServer(
		sSrvNetId:= , 
		sLocalHost:=sHost , 
		nLocalPort:=nPort , 
		bStartConnect:=bEnable , 
		tcpipSDataLen:=TO_UDINT(LEN(tcpipSendDataBuff_Server)) , 
		tcpipSData:=ADR(tcpipSendDataBuff_Server) , 
		bSend:= , 
		tcpipRecDataLen:=SIZEOF(tcpipRecDataBuff_Server) , 
		tcpipRecData:=ADR(tcpipRecDataBuff_Server) , 
		bAccepted=> , 
		bSendBusy=> , 
		bRecData=> );
	bSendCondition:=tcpipServer.bAccepted AND NOT tcpipServer.bSendBusy;
	//TCPIP连接
	bSocketConnected:=tcpipServer.bAccepted;
	IF NOT tcpipServer.bAccepted THEN
		length:=0;
		endPoint:=cNumBegin;
	END_IF
	tcpConnectR_Trig(CLK:=tcpipServer.bAccepted);
	tcpConnectF_Trig(CLK:=tcpipServer.bAccepted);

1://TCPIP client
	tcpipClient(
		sSrvNetId:= , 
		sRemoteHost:=sHost , 
		nRemotePort:=nPort , 
		bStartConnect:=bEnable , 
		tcpipSDataLen:=TO_UDINT(LEN(tcpipSendDataBuff_Client)) , 
		tcpipSData:=ADR(tcpipSendDataBuff_Client) , 
		bSend:= , 
		tcpipRecDataLen:=SIZEOF(tcpipRecDataBuff_Client) , 
		tcpipRecData:=ADR(tcpipRecDataBuff_Client) , 
		bConnected=> , 
		bSendBusy=> , 
		bRecData=> );
	bSendCondition:=tcpipClient.bConnected AND NOT tcpipClient.bSendBusy;
	//TCPIP连接
	bSocketConnected:=tcpipClient.bConnected;
	IF NOT tcpipClient.bConnected THEN
		length:=0;
		endPoint:=cNumBegin;
	END_IF
	tcpConnectR_Trig(CLK:=tcpipClient.bConnected);
	tcpConnectF_Trig(CLK:=tcpipClient.bConnected);
END_CASE

IF tcpConnectR_Trig.Q THEN
	FOR logHandleArray_index:=1 TO logHandleArrayLength DO
		logHandleArray[logHandleArray_index]^.append(CONCAT(sTerminalName, ' has been connected'));
	END_FOR
	registerStep:=10;
END_IF
IF tcpConnectF_Trig.Q THEN
	FOR logHandleArray_index:=1 TO logHandleArrayLength DO
		logHandleArray[logHandleArray_index]^.append(CONCAT(sTerminalName, ' has been disconnected'));
	END_FOR
	registerStep:=0;
END_IF
//数据接收处理
CASE nSocketType OF
0://TCPIP server
	IF tcpipServer.bRecData THEN
		tcpipRecData:=tcpipRecDataBuff_Server;//buff转存
		tcpipRecDataBuff_Server:=tcpipRecDataClear;//转存之后清空buff
		dataProcessing();
	END_IF
1://TCPIP client
	IF tcpipClient.bRecData THEN
		tcpipRecData:=tcpipRecDataBuff_Client;//buff转存
		tcpipRecDataBuff_Client:=tcpipRecDataClear;//转存之后清空buff
		dataProcessing();
	END_IF
END_CASE


popup();

CASE registerStep OF
0:
	//Ready
END_CASE

METHOD appendSend : BOOL
VAR_INPUT
	str			:STRING(255);
END_VAR
VAR
	suffix					:STRING;
	strTemp_appendSend		:STRING(255);
END_VAR

IF endPoint>(cNumEnd-1) THEN
	RETURN;
END_IF
suffix:=sSendSuffix;//此处可统一添加发送后缀字符 $R$N

strTemp_appendSend:=CONCAT(str,suffix);
sendDataArray[endPoint]:=strTemp_appendSend;

endPoint:=endPoint+1;
length:=endPoint-cNumBegin;
END_METHOD

METHOD dataProcessing : BOOL
VAR_INPUT
END_VAR
FOR logHandleArray_index:=1 TO logHandleArrayLength DO
	CASE nSocketType OF
	0://TCPIP server
		logHandleArray[logHandleArray_index]^.append(CONCAT(CONCAT(CONCAT('Recevie From ', sTerminalName), ' -- '),tcpipRecData));
	1://TCPIP client
		logHandleArray[logHandleArray_index]^.append(CONCAT(CONCAT(CONCAT('Recevie From ', sTerminalName), ' -- '),tcpipRecData));
	END_CASE
END_FOR

appendSend(tcpipRecData);
IF FIND(tcpipRecData, 'FASDFASDD')>0 THEN
	;
END_IF
END_METHOD

